FUNCTION "TE-SS" : VOID	// FC 11
AUTHOR : SIMATIC
FAMILY : EA_DIS
NAME : TE_SS
VERSION : 3.0
BEGIN
// (block stored without names or comments; labels and parameter names are numbered)
NETWORK
TITLE =
      L     0;
      L     #PARAM22;
      ==I;
      JC    M001;
      T     MW 214;
      L     MB 214;
      T     LW 10;
      OPN   DB [LW 10];
      L     MB 215;
      SLW   3;
      LAR1;
      L     DBW [AR1,P#0.0];
      T     MB 227;
M001: L     #PARAM20;
      T     MW 214;
      L     MB 214;
      T     LW 10;
      OPN   DB [LW 10];
      L     #PARAM20;
      T     MW 214;
      L     MB 215;
      SLW   3;
      LAR1;
      L     DBW [AR1,P#0.0];
      T     MW 200;
      L     DBW [AR1,P#2.0];
      T     MW 202;
      L     DBW [AR1,P#4.0];
      T     MW 204;
      L     DBW [AR1,P#10.0];
      T     MW 208;
      L     DBW [AR1,P#12.0];
      T     MW 210;
      L     DBW [AR1,P#14.0];
      T     MW 212;
      L     DBW [AR1,P#16.0];
      T     MW 206;
      A     #PARAM1;
      A     M 204.7;
      =     M 203.2;
      A     #PARAM1;
      AN    M 204.7;
      =     M 202.0;
      A     #PARAM2;
      =     M 202.1;
      A     #PARAM3;
      AN    M 203.3;
      =     M 211.5;
      A     #PARAM3;
      =     M 203.3;
      A     #PARAM4;
      AN    M 203.0;
      =     M 211.7;
      A     #PARAM4;
      =     M 203.0;
      A     #PARAM8;
      AN    M 203.1;
      =     M 211.6;
      A     #PARAM8;
      =     M 203.1;
      A     #PARAM9;
      AN    M 203.4;
      =     M 211.4;
      A     #PARAM9;
      =     M 203.4;
      A     #PARAM10;
      =     M 202.2;
      A     #PARAM11;
      =     M 203.5;
      A     #PARAM7;
      =     M 213.0;
      A     #PARAM6;
      =     M 210.1;
      A     #PARAM13;
      =     M 210.7;
      A     #PARAM14;
      =     M 210.6;
      A     #PARAM15;
      =     M 210.5;
      A     #PARAM16;
      =     M 210.4;
      A     #PARAM17;
      =     M 210.3;
      A     #PARAM18;
      =     M 210.2;
      A     #PARAM19;
      =     M 200.4;
      A     #PARAM12;
      =     M 210.0;
      A     #PARAM5;
      =     M 203.6;
NETWORK
TITLE =
      A     M 210.7;
      AN    M 210.6;
      =     M 212.7;
      AN    M 210.7;
      A     M 210.6;
      =     M 212.5;
      A     M 210.5;
      AN    M 210.4;
      =     M 212.6;
      AN    M 210.5;
      A     M 210.4;
      =     M 212.4;
NETWORK
TITLE =
      A     M 227.3;
      AN    M 202.5;
      =     M 211.3;
      A     M 227.3;
      =     M 202.5;
      A     M 227.2;
      AN    M 202.6;
      =     M 211.2;
      A     M 227.2;
      =     M 202.6;
NETWORK
TITLE =
      A     M 203.1;
      A     M 210.1;
      AN    M 203.0;
      AN    M 203.6;
      =     M 218.7;
      A     M 203.0;
      A     M 210.1;
      AN    M 203.6;
      =     M 219.7;
      A     M 227.2;
      A     M 227.1;
      AN    M 227.3;
      AN    M 227.0;
      AN    M 219.7;
      AN    M 203.6;
      =     M 218.5;
      A     M 227.3;
      A     M 227.1;
      AN    M 227.0;
      AN    M 218.7;
      AN    M 203.6;
      =     M 219.5;
      A     M 203.4;
      AN    M 203.3;
      AN    M 219.7;
      AN    M 203.6;
      AN    M 227.0;
      AN    M 219.5;
      =     M 218.3;
      A     M 203.3;
      AN    M 218.7;
      AN    M 218.5;
      AN    M 203.6;
      AN    M 227.0;
      =     M 219.3;
      A     M 218.7;
      O     M 218.5;
      O     M 218.3;
      =     M 212.3;
      A     M 219.7;
      O     M 219.5;
      O     M 219.3;
      =     M 212.1;
      A     M 211.6;
      A     M 218.7;
      O;
      A     M 211.2;
      A     M 218.5;
      O;
      A     M 211.4;
      A     M 218.3;
      =     M 212.2;
      A     M 211.7;
      A     M 219.7;
      O;
      A     M 211.3;
      A     M 219.5;
      O;
      A     M 211.5;
      A     M 219.3;
      =     M 212.0;
NETWORK
TITLE =
      A     M 211.6;
      O     M 211.2;
      =     M 213.4;
      A     M 211.7;
      O     M 211.3;
      =     M 213.5;
      A     M 203.6;
      O     M 227.0;
      =     M 213.7;
NETWORK
TITLE =
      A     M 212.7;
      O     M 213.7;
      O     M 212.3;
      R     M 211.1;
      R     M 211.0;
      A     M 203.2;
      S     M 211.1;
      A     M 202.0;
      S     M 211.0;
      A     M 212.6;
      O     M 213.7;
      O     M 212.1;
      R     M 213.1;
      A     M 203.5;
      S     M 213.1;
NETWORK
TITLE =
      A     M 203.1;
      A     M 210.1;
      O(;
      A     M 227.2;
      A     M 227.1;
      );
      O     M 203.4;
      =     M 213.2;
      A     M 203.0;
      A     M 210.1;
      O(;
      A     M 227.3;
      A     M 227.1;
      );
      O     M 203.3;
      =     M 213.3;
      A     M 213.2;
      O     M 203.5;
      ON    M 202.1;
      A     M 213.3;
      A     M 212.5;
      O(;
      A     M 213.3;
      O     M 203.2;
      O     M 202.0;
      ON    M 202.2;
      A     M 213.2;
      A     M 212.4;
      );
      O(;
      A     M 203.2;
      O     M 202.0;
      A     M 203.5;
      A     M 212.5;
      );
      =     M 201.1;
NETWORK
TITLE =
      L     0;
      L     MW 206;
      >=I;
      JC    M002;
      AN    "M 1.3";
      JC    M002;
      L     MW 206;
      L     1;
      -I;
      T     MW 206;
      L     MB 207;
      T     DBW [AR1,P#16.0];
M002: NOP   0;
NETWORK
TITLE =
      L     MB 205;
      T     MB 209;
      L     0;
      >I;
      JC    M006;
      A     M 212.7;
      A     M 212.4;
      AN    M 204.5;
      O;
      A     M 212.7;
      A     M 212.4;
      A     M 204.5;
      AN    M 210.3;
      L     1;
      JC    M005;
      A     M 212.6;
      A     M 212.5;
      AN    M 204.6;
      O;
      A     M 212.6;
      A     M 212.5;
      A     M 204.6;
      AN    M 210.2;
      L     9;
      JC    M005;
      A     M 212.0;
      A     M 202.1;
      AN    M 213.1;
      O     M 211.1;
      O     M 211.0;
      L     10;
      JC    M003;
      AN    M 212.2;
      ON    M 202.2;
      AN    M 213.1;
      JC    M004;
      L     2;
M003: T     MB 209;
      L     DBW [AR1,P#6.0];
      T     MW 206;
      L     MW 206;
      T     DBW [AR1,P#16.0];
      JU    M006;
M004: L     0;
M005: T     MB 209;
M006: NOP   0;
NETWORK
TITLE =
      L     MB 205;
      L     1;
      <>I;
      JC    M008;
      A     M 212.6;
      O     M 212.5;
      L     14;
      JC    M007;
      A     M 211.0;
      O     M 211.1;
      JC    M008;
      AN    M 212.2;
      ON    M 202.2;
      AN    M 213.1;
      JC    M008;
      L     DBW [AR1,P#6.0];
      T     MW 206;
      L     MW 206;
      T     DBW [AR1,P#16.0];
      L     2;
M007: T     MB 209;
M008: NOP   0;
NETWORK
TITLE =
      L     MB 205;
      L     2;
      <>I;
      JC    M014;
      A     M 212.0;
      A     M 202.1;
      AN    M 213.1;
      O     M 211.0;
      O     M 211.1;
      L     12;
      JC    M009;
      A     M 212.5;
      L     4;
      JC    M012;
      A     M 213.7;
      AN    M 213.1;
      O     M 200.4;
      O;
      AN    M 212.3;
      AN    M 213.0;
      AN    M 213.1;
      L     0;
      JC    M013;
      AN    M 210.2;
      L     6;
      JC    M013;
      L     MW 206;
      L     0;
      <>I;
      JC    M014;
      L     3;
      T     MB 209;
      JU    M014;
M009: T     MB 209;
      L     DBW [AR1,P#6.0];
      JU    M011;
M010: L     DBW [AR1,P#8.0];
M011: T     MW 206;
      T     DBW [AR1,P#16.0];
      JU    M014;
M012: T     MB 209;
      JU    M010;
M013: T     MB 209;
      L     0;
      JU    M011;
M014: NOP   0;
NETWORK
TITLE =
      L     MB 205;
      L     3;
      <>I;
      JC    M017;
      A     M 211.1;
      O     M 200.4;
      O;
      A     M 213.7;
      AN    M 213.1;
      O;
      AN    M 213.0;
      AN    M 212.3;
      AN    M 213.1;
      O;
      A     M 212.0;
      A     M 202.1;
      AN    M 213.1;
      L     0;
      JC    M016;
      A     M 212.7;
      A     M 213.5;
      L     1;
      JC    M016;
      A     M 212.5;
      A     M 213.4;
      L     4;
      JC    M015;
      A     M 210.2;
      L     6;
      JC    M017;
M015: T     MB 209;
      L     DBW [AR1,P#8.0];
      T     MW 206;
      L     MW 206;
      T     DBW [AR1,P#16.0];
      JU    M017;
M016: T     MB 209;
M017: NOP   0;
NETWORK
TITLE =
      L     MB 205;
      L     4;
      <>I;
      JC    M021;
      A     M 212.0;
      A     M 202.1;
      AN    M 213.1;
      O     M 211.0;
      O     M 211.1;
      L     10;
      JC    M018;
      A     M 212.6;
      AN    M 204.6;
      O;
      A     M 212.6;
      A     M 204.6;
      AN    M 210.2;
      L     9;
      JC    M020;
      A     M 213.7;
      AN    M 213.1;
      O     M 200.4;
      O;
      AN    M 212.3;
      AN    M 213.0;
      AN    M 213.1;
      L     0;
      JC    M020;
      AN    M 210.2;
      L     6;
      JC    M020;
      L     MW 206;
      L     0;
      <>I;
      JC    M021;
      L     5;
      T     MB 209;
      JU    M021;
M018: T     MB 209;
      L     DBW [AR1,P#6.0];
M019: T     MW 206;
      L     MW 206;
      T     DBW [AR1,P#16.0];
      JU    M021;
M020: T     MB 209;
      L     0;
      JU    M019;
M021: NOP   0;
NETWORK
TITLE =
      L     MB 205;
      L     5;
      <>I;
      JC    M024;
      A     M 213.7;
      O     M 200.4;
      O;
      AN    M 213.0;
      AN    M 212.3;
      AN    M 213.1;
      L     0;
      JC    M023;
      A     M 212.6;
      AN    M 204.6;
      A     M 213.4;
      O;
      A     M 212.6;
      A     M 204.6;
      AN    M 210.2;
      A     M 213.4;
      L     9;
      JC    M023;
      A     M 211.1;
      O;
      A     M 212.0;
      A     M 202.1;
      AN    M 213.1;
      L     10;
      JC    M022;
      A     M 210.2;
      L     6;
      JC    M024;
M022: T     MB 209;
      L     DBW [AR1,P#6.0];
      T     MW 206;
      L     MW 206;
      T     DBW [AR1,P#16.0];
      JU    M024;
M023: T     MB 209;
M024: NOP   0;
NETWORK
TITLE =
      L     MB 205;
      L     6;
      <>I;
      JC    M025;
      AN    M 213.5;
      AN    M 213.4;
      L     0;
      JC    M025;
      T     MB 209;
M025: NOP   0;
NETWORK
TITLE =
      L     MB 205;
      L     9;
      <>I;
      JC    M027;
      A     M 212.7;
      O     M 212.4;
      O     M 200.4;
      L     6;
      JC    M026;
      AN    M 211.0;
      AN    M 211.1;
      A(;
      AN    M 212.0;
      ON    M 202.1;
      O     M 213.1;
      );
      JC    M027;
      L     DBW [AR1,P#6.0];
      T     MW 206;
      L     MW 206;
      T     DBW [AR1,P#0.0];
      L     10;
M026: T     MB 209;
M027: NOP   0;
NETWORK
TITLE =
      L     MB 205;
      L     10;
      <>I;
      JC    M033;
      A     M 212.2;
      A     M 202.2;
      O     M 213.1;
      AN    M 211.0;
      AN    M 211.1;
      L     4;
      JC    M028;
      A     M 212.4;
      L     12;
      JC    M031;
      A     M 213.7;
      AN    M 211.1;
      AN    M 211.0;
      O     M 200.4;
      O;
      AN    M 212.1;
      AN    M 213.0;
      AN    M 211.1;
      AN    M 211.0;
      L     0;
      JC    M032;
      AN    M 210.3;
      L     14;
      JC    M032;
      L     MW 206;
      L     0;
      <>I;
      JC    M033;
      L     11;
      T     MB 209;
      JU    M033;
M028: T     MB 209;
      L     DBW [AR1,P#6.0];
      JU    M030;
M029: L     DBW [AR1,P#8.0];
M030: T     MW 206;
      L     MW 206;
      T     DBW [AR1,P#16.0];
      JU    M033;
M031: T     MB 209;
      JU    M029;
M032: T     MB 209;
      L     0;
      JU    M030;
M033: NOP   0;
NETWORK
TITLE =
      L     MB 205;
      L     11;
      <>I;
      JC    M036;
      A     M 200.4;
      O;
      A     M 213.7;
      AN    M 211.1;
      AN    M 211.0;
      O;
      AN    M 213.0;
      AN    M 212.1;
      AN    M 211.1;
      AN    M 211.0;
      O;
      A     M 212.2;
      A     M 202.2;
      AN    M 211.1;
      AN    M 211.0;
      L     0;
      JC    M035;
      A     M 212.6;
      A     M 213.4;
      L     9;
      JC    M035;
      A     M 212.4;
      A     M 213.5;
      L     12;
      JC    M034;
      A     M 210.3;
      L     14;
      JC    M036;
M034: T     MB 209;
      L     DBW [AR1,P#8.0];
      T     MW 206;
      L     MW 206;
      T     DBW [AR1,P#16.0];
      JU    M036;
M035: T     MB 209;
M036: NOP   0;
NETWORK
TITLE =
      L     MB 205;
      L     12;
      <>I;
      JC    M040;
      A     M 212.2;
      A     M 202.2;
      O     M 213.1;
      AN    M 211.0;
      AN    M 211.1;
      L     2;
      JC    M037;
      A     M 212.7;
      AN    M 204.5;
      O;
      A     M 212.7;
      A     M 204.5;
      AN    M 210.3;
      =     M 228.0;
      A     M 228.0;
      A     M 211.1;
      L     6;
      JC    M039;
      A     M 228.0;
      L     1;
      JC    M039;
      A     M 213.7;
      AN    M 211.1;
      AN    M 211.0;
      O     M 200.4;
      O;
      AN    M 212.1;
      AN    M 213.0;
      AN    M 211.1;
      AN    M 211.0;
      L     0;
      JC    M039;
      AN    M 210.3;
      L     14;
      JC    M039;
      L     MW 206;
      L     0;
      <>I;
      JC    M040;
      L     13;
      T     MB 209;
      JU    M040;
M037: T     MB 209;
      L     DBW [AR1,P#6.0];
M038: T     MW 206;
      L     MW 206;
      T     DBW [AR1,P#16.0];
      JU    M040;
M039: T     MB 209;
      L     0;
      JU    M038;
M040: NOP   0;
NETWORK
TITLE =
      L     MB 205;
      L     13;
      <>I;
      JC    M043;
      A     M 213.7;
      O     M 200.4;
      O;
      AN    M 213.0;
      AN    M 212.1;
      AN    M 211.1;
      AN    M 211.0;
      L     0;
      JC    M042;
      A     M 212.7;
      AN    M 204.5;
      A     M 213.5;
      O;
      A     M 212.7;
      A     M 204.5;
      AN    M 210.3;
      A     M 213.5;
      L     1;
      JC    M042;
      A     M 212.2;
      A     M 202.2;
      AN    M 211.1;
      AN    M 211.0;
      L     2;
      JC    M041;
      A     M 210.3;
      L     14;
      JC    M043;
M041: T     MB 209;
      L     DBW [AR1,P#6.0];
      T     MW 206;
      L     MW 206;
      T     DBW [AR1,P#16.0];
      JU    M043;
M042: T     MB 209;
M043: NOP   0;
NETWORK
TITLE =
      L     MB 205;
      L     14;
      <>I;
      JC    M044;
      AN    M 213.5;
      AN    M 213.4;
      L     0;
      JC    M044;
      T     MB 209;
M044: NOP   0;
NETWORK
TITLE =
      L     MB 209;
      T     MB 205;
      L     15;
      <I;
      A(;
      +     -7;
      <>I;
      );
      A(;
      +     -1;
      <>I;
      );
      AN    "M 0.7";
      JC    M045;
      L     0;
      T     MB 205;
M045: NOP   0;
NETWORK
TITLE =
      A     M 212.6;
      A     M 212.7;
      O;
      AN    M 212.6;
      AN    M 212.4;
      O;
      AN    M 212.7;
      AN    M 212.5;
      =     M 200.7;
      AN    M 210.2;
      AN    M 210.3;
      =     M 202.7;
      A     M 212.6;
      AN    M 210.2;
      =     M 200.5;
      A     M 212.7;
      AN    M 210.3;
      =     M 200.6;
      AN    M 209.0;
      A     M 209.1;
      A     M 209.2;
      AN    M 200.7;
      =     M 228.0;
      AN    M 209.3;
      A     M 228.0;
      =     M 200.2;
      A     M 209.3;
      A     M 228.0;
      =     M 200.3;
      A     M 209.0;
      A(;
      A     M 209.1;
      AN    M 209.2;
      O;
      AN    M 209.1;
      A     M 209.2;
      );
      AN    M 200.7;
      AN    M 202.7;
      =     M 228.0;
      A     M 228.0;
      AN    M 209.3;
      =     M 200.1;
      A     M 228.0;
      A     M 209.3;
      =     M 200.0;
NETWORK
TITLE =
      A     M 201.1;
      =     M 203.7;
      A     M 209.0;
      A     M 209.1;
      A     M 209.2;
      O     M 200.4;
      O     M 200.3;
      O     M 200.2;
      O     M 200.1;
      O     M 200.0;
      O     M 200.7;
      O     M 202.7;
      =     M 201.0;
      A(;
      A     M 209.1;
      AN    M 209.2;
      O;
      AN    M 209.1;
      A     M 209.2;
      );
      AN    M 209.0;
      =     M 228.0;
      A     M 228.0;
      A     M 209.3;
      =     M 201.4;
      A     M 200.0;
      O     M 200.3;
      AN    M 200.7;
      AN    M 202.7;
      =     M 201.2;
      A     M 212.7;
      AN    M 204.5;
      O;
      A     M 212.7;
      A     M 204.5;
      AN    M 210.3;
      =     M 201.3;
      =     M 202.4;
      =     #PARAM24;
      A     M 228.0;
      AN    M 209.3;
      =     M 201.7;
      A     M 200.1;
      O     M 200.2;
      AN    M 200.7;
      AN    M 202.7;
      =     M 201.5;
      A     M 212.6;
      AN    M 204.6;
      O;
      A     M 212.6;
      AN    M 210.2;
      A     M 204.6;
      =     M 201.6;
      =     M 202.3;
      =     #PARAM25;
NETWORK
TITLE =
      A     M 201.0;
      O     M 203.7;
      AN    M 201.1;
      =     #PARAM26;
      A     M 201.0;
      A     "M 1.6";
      O     M 203.7;
      O     #PARAM12;
      =     #PARAM29;
      A     M 201.7;
      A     "M 1.5";
      O;
      A     M 201.5;
      A     "M 1.6";
      O     M 201.6;
      O     #PARAM12;
      =     #PARAM28;
      A     M 201.4;
      A     "M 1.5";
      O;
      A     M 201.2;
      A     "M 1.6";
      O     M 201.3;
      O     #PARAM12;
      =     #PARAM27;
NETWORK
TITLE =
      A(;
      A     M 209.1;
      AN    M 209.2;
      O;
      AN    M 209.1;
      A     M 209.2;
      );
      AN    M 209.3;
      =     #PARAM31;
      A(;
      A     M 209.1;
      AN    M 209.2;
      O;
      AN    M 209.1;
      A     M 209.2;
      );
      A     M 209.3;
      =     #PARAM30;
      L     MW 200;
      T     DBW [AR1,P#0.0];
      L     MW 202;
      T     DBW [AR1,P#2.0];
      L     MW 204;
      T     DBW [AR1,P#4.0];
      L     MW 208;
      T     DBW [AR1,P#10.0];
      L     MW 210;
      T     DBW [AR1,P#12.0];
      L     MW 212;
      T     DBW [AR1,P#14.0];
      L     MW 206;
      T     DBW [AR1,P#16.0];
      L     0;
      L     #PARAM23;
      ==I;
      JC    M048;
      T     MW 216;
      T     MW 240;
      L     MB 216;
      SLW   3;
      LAR1;
      L     DBW [AR1,P#0.0];
      T     MW 242;
      L     MW 240;
      SLW   12;
      SRW   12;
      T     MW 240;
      L     8;
      L     MB 241;
      >I;
      JC    M046;
      +     -8;
      SLW   8;
      INC   242;
      JU    M047;
M046: SLW   8;
      INC   243;
M047: T     MW 244;
      L     MB 244;
      L     MB 245;
      SLW   3;
      OW;
      LAR2;
      A     M 201.0;
      O     M 203.3;
      =     M [AR2,P#0.0];
      L     MB 217;
      SLW   3;
      LAR1;
      L     MW 242;
      T     DBW [AR1,P#0.0];
M048: L     0;
      L     #PARAM21;
      ==I;
      BEC;
      T     MW 216;
      L     MB 216;
      T     LW 10;
      OPN   DB [LW 10];
      L     MB 217;
      SLW   3;
      LAR1;
      L     MW 200;
      T     DBW [AR1,P#0.0];
      L     MW 202;
      T     DBW [AR1,P#2.0];
END_FUNCTION

FUNCTION "TE-REK" : VOID	// FC 12
AUTHOR : SIMATIC
FAMILY : SIMATIC
NAME : TE_REK
VERSION : 3.0
BEGIN
// (block stored without names or comments; labels and parameter names are numbered)
NETWORK
TITLE =
      L     0;
      L     #PARAM20;
      ==I;
      JC    M001;
      T     MW 212;
      L     MB 212;
      T     LW 10;
      OPN   DB [LW 10];
      L     MB 213;
      SLW   3;
      LAR1;
      L     DBW [AR1,P#2.0];
M001: T     MW 210;
      L     #PARAM18;
      T     MW 214;
      L     MB 214;
      T     LW 10;
      OPN   DB [LW 10];
      L     MB 215;
      SLW   3;
      LAR1;
      L     DBW [AR1,P#0.0];
      T     MW 200;
      L     DBW [AR1,P#2.0];
      T     MW 202;
      A     #PARAM1;
      =     M 203.1;
      A     #PARAM2;
      =     M 200.4;
      A     #PARAM3;
      AN    M 202.7;
      =     M 210.0;
      A     #PARAM3;
      =     M 202.7;
      A     #PARAM4;
      AN    M 200.2;
      =     M 210.1;
      A     #PARAM4;
      =     M 200.2;
      A     #PARAM6;
      AN    M 200.3;
      =     M 210.3;
      A     #PARAM6;
      =     M 200.3;
      A     #PARAM7;
      AN    M 202.6;
      =     M 210.2;
      A     #PARAM7;
      =     M 202.6;
      A     #PARAM8;
      =     M 200.5;
      A     #PARAM9;
      =     M 203.0;
      A     #PARAM10;
      =     M 210.7;
      A     #PARAM5;
      =     M 202.5;
      A     #PARAM11;
      AN    M 200.0;
      =     M 210.4;
      A     #PARAM11;
      =     M 200.0;
      A     #PARAM12;
      AN    M 200.1;
      =     M 210.5;
      A     #PARAM12;
      =     M 200.1;
      A     #PARAM13;
      AN    M 202.4;
      =     M 210.6;
      A     #PARAM13;
      =     M 202.4;
      AN    #PARAM14;
      =     M 200.6;
      A     #PARAM15;
      =     M 203.3;
NETWORK
TITLE =
      A     M 211.0;
      AN    M 202.3;
      =     M 211.5;
      A     M 211.0;
      =     M 202.3;
      A     M 211.2;
      AN    M 202.1;
      =     M 211.6;
      A     M 211.2;
      =     M 202.1;
      A     M 211.3;
      AN    M 202.2;
      =     M 211.7;
      A     M 211.3;
      =     M 202.2;
NETWORK
TITLE =
      AN    M 200.7;
      AN    M 201.5;
      S     M 200.7;
      A     "´1´";
      R     M 201.7;
      R     M 201.6;
NETWORK
TITLE =
      A     M 202.7;
      A     M 202.5;
      O;
      A     M 202.1;
      A     M 211.1;
      O;
      A     M 200.2;
      =     M 202.0;
      A     M 202.6;
      A     M 202.5;
      O;
      A     M 202.2;
      A     M 211.1;
      O;
      A     M 200.3;
      =     M 203.6;
NETWORK
TITLE =
      AN    M 200.7;
      JC    M005;
      AN    M 203.1;
      JC    M002;
      L     MW 214;
      +     5;
      T     MW 216;
      +     -2;
      T     MW 218;
      L     DBW [AR1,P#10.0];
      T     DBW [AR1,P#6.0];
      JU    M005;
M002: AN    M 203.0;
      JC    M003;
      L     MW 214;
      +     6;
      T     MW 216;
      +     -3;
      T     MW 218;
      L     DBW [AR1,P#12.0];
      T     DBW [AR1,P#6.0];
      JU    M008;
M003: A     M 211.5;
      A     M 211.1;
      AN    M 202.4;
      O;
      A     M 210.6;
      A     M 202.5;
      AN    M 211.0;
      S     M 201.7;
      A     M 210.5;
      AN    M 200.0;
      O     M 201.7;
      O     M 211.5;
      R     M 200.7;
      S     M 201.5;
      R     M 210.5;
      R     M 211.5;
      R     M 210.6;
      A     M 202.0;
      AN    M 203.6;
      A     M 200.4;
      S     M 203.5;
      AN    M 202.0;
      R     M 203.5;
      A     M 203.6;
      AN    M 202.0;
      A     M 200.5;
      S     M 203.4;
      AN    M 203.6;
      R     M 203.4;
      AN    M 203.5;
      JC    M006;
      L     MW 214;
      +     2;
      T     MW 216;
      L     DBW [AR1,P#4.0];
      T     MW 206;
      SLW   6;
      SRW   6;
      L     DBB [AR1,P#4.0];
      SRW   2;
      +I;
      L     1000;
      TAK;
      >I;
      JC    M004;
      TAK;
M004: T     MW 204;
      L     MB 206;
      SRW   2;
      SLW   10;
      OW;
      T     DBW [AR1,P#4.0];
      L     MW 214;
      +     3;
      T     MW 216;
      L     DBW [AR1,P#6.0];
      L     MW 204;
      -I;
      T     DBW [AR1,P#6.0];
M005: JU    M008;
M006: AN    M 203.4;
      JC    M009;
      L     MW 214;
      +     2;
      T     MW 216;
      L     DBW [AR1,P#4.0];
      T     MW 206;
      SLW   6;
      SRW   6;
      L     DBB [AR1,P#4.0];
      SRW   2;
      +I;
      L     1000;
      TAK;
      >I;
      JC    M007;
      TAK;
M007: T     MW 204;
      L     MB 206;
      SRW   2;
      SLW   10;
      OW;
      T     DBW [AR1,P#4.0];
      L     MW 214;
      +     3;
      T     MW 216;
      L     DBW [AR1,P#6.0];
      L     MW 204;
      +I;
      T     DBW [AR1,P#6.0];
M008: JU    M010;
M009: L     MW 214;
      +     2;
      T     MW 216;
      L     DBB [AR1,P#4.0];
      SRW   2;
      SLW   10;
      T     DBW [AR1,P#4.0];
      L     0;
      L     #PARAM20;
      ==I;
      JC    M010;
      T     MW 212;
      L     MW 214;
      +     8;
      T     MW 216;
      L     DBW [AR1,P#16.0];
      T     LD 0;
      L     MB 212;
      T     LW 10;
      OPN   DB [LW 10];
      L     MB 213;
      SLW   3;
      LAR1;
      L     LD 0;
      L     DBW [AR1,P#0.0];
      ==I;
      T     LD 0;
      L     MB 214;
      T     LW 10;
      OPN   DB [LW 10];
      JC    M010;
      L     MB 215;
      SLW   3;
      LAR1;
      L     LD 0;
      T     DBW [AR1,P#16.0];
      L     MW 214;
      +     3;
      T     MW 216;
      L     LD 0;
      T     DBW [AR1,P#6.0];
M010: NOP   0;
NETWORK
TITLE =
      AN    M 201.5;
      JC    M013;
      AN    M 203.1;
      JC    M011;
      L     MW 214;
      +     5;
      T     MW 216;
      +     -2;
      T     MW 218;
      L     MB 215;
      SLW   3;
      LAR1;
      L     DBW [AR1,P#10.0];
      T     DBW [AR1,P#6.0];
      JU    M012;
M011: AN    M 203.0;
      JC    M012;
      L     MW 214;
      +     6;
      T     MW 216;
      +     -3;
      T     MW 218;
      L     MB 215;
      SLW   3;
      LAR1;
      L     DBW [AR1,P#12.0];
      T     DBW [AR1,P#6.0];
M012: A     M 211.5;
      A     M 211.1;
      AN    M 202.4;
      O;
      A     M 210.6;
      A     M 202.5;
      AN    M 211.0;
      S     M 201.6;
      A     M 210.4;
      AN    M 200.1;
      AN    M 202.4;
      AN    M 202.3;
      O     M 211.5;
      O     M 201.6;
      O     M 200.6;
      O     "M 0.6";
      O     M 203.3;
      S     M 200.7;
      R     M 201.5;
      A     M 200.7;
      O     M 203.0;
      O     M 203.1;
      JC    M013;
      L     #PARAM16;
      T     MW 216;
      L     MB 216;
      T     LW 10;
      OPN   DB [LW 10];
      L     MB 217;
      SLW   3;
      LAR1;
      L     DBD [AR1,P#0.0];
      T     LD 0;
      L     MB 214;
      T     LW 10;
      OPN   DB [LW 10];
      L     MW 214;
      +     3;
      T     MW 216;
      L     MB 215;
      SLW   3;
      LAR1;
      L     LW 8;
      L     LD 0;
      T     DBD [AR1,P#18.0];
M013: NOP   0;
NETWORK
TITLE =
      L     MW 214;
      +     3;
      T     MW 216;
      +     4;
      T     MW 218;
      L     MB 215;
      SLW   3;
      LAR1;
      L     DBW [AR1,P#6.0];
      L     DBW [AR1,P#14.0];
      ==I;
      T     MW 222;
      JC    M019;
      <=I;
      JC    M016;
      AN    M 200.5;
      AN    M 203.0;
      JC    M019;
      TAK;
      T     MW 224;
      L     MW 214;
      +     6;
      T     MW 216;
      L     DBW [AR1,P#12.0];
      L     DBW [AR1,P#10.0];
      -I;
      SRW   3;
      L     MW 222;
      +I;
      L     MW 224;
      <=I;
      TAK;
      JC    M014;
      TAK;
M014: T     MW 222;
      L     MW 214;
      +     6;
      T     MW 216;
      L     DBW [AR1,P#12.0];
      L     MW 222;
      >I;
      JC    M015;
      L     MW 214;
      +     3;
      T     MW 216;
      L     DBW [AR1,P#12.0];
      T     DBW [AR1,P#6.0];
M015: NOP   0;
      T     DBW [AR1,P#14.0];
      T     MW 222;
      L     MW 218;
      +     2;
      T     MW 218;
      TAK;
      L     MW 222;
      L     1;
      *I;
      DTR;
      T     DBD [AR1,P#18.0];
      JU    M019;
M016: ==I;
      JC    M019;
      AN    M 200.4;
      AN    M 203.1;
      JC    M019;
      TAK;
      T     MW 224;
      L     MW 214;
      +     6;
      T     MW 216;
      L     DBW [AR1,P#12.0];
      L     DBW [AR1,P#10.0];
      -I;
      SRW   3;
      L     MW 222;
      TAK;
      -I;
      L     MW 224;
      >=I;
      TAK;
      JC    M017;
      TAK;
M017: T     MW 222;
      L     MW 214;
      +     5;
      T     MW 216;
      L     DBW [AR1,P#10.0];
      L     MW 222;
      <I;
      JC    M018;
      L     MW 214;
      +     3;
      T     MW 216;
      L     DBW [AR1,P#10.0];
      T     DBW [AR1,P#6.0];
M018: NOP   0;
      T     DBW [AR1,P#14.0];
      T     MW 222;
      L     1;
      *I;
      DTR;
      T     DBD [AR1,P#18.0];
M019: NOP   0;
NETWORK
TITLE =
      A(;
      A     M 203.0;
      O     M 203.1;
      ON    M 200.5;
      ON    M 200.4;
      A     M 201.5;
      );
      O(;
      A(;
      O     M 202.4;
      O     M 202.3;
      );
      A(;
      O     M 200.6;
      O     M 203.3;
      );
      );
      O(;
      A     M 203.0;
      ON    M 200.4;
      A     M 202.0;
      A     M 200.7;
      );
      O(;
      A     M 203.1;
      ON    M 200.5;
      A     M 203.6;
      A     M 200.7;
      );
      =     M 201.3;
      A     M 203.5;
      O     M 203.4;
      O     M 203.0;
      O     M 203.1;
      =     M 203.7;
      =     M 203.2;
NETWORK
TITLE =
// (network holds code this reader does not know; not shown)
END_FUNCTION

FUNCTION "TE-TS" : VOID	// FC 13
AUTHOR : SIMATIC
FAMILY : EA_DIS
NAME : TE_TS
VERSION : 3.0
BEGIN
// (block stored without names or comments; labels and parameter names are numbered)
NETWORK
TITLE =
      L     0;
      L     #PARAM9;
      ==I;
      JC    M001;
      T     MW 212;
      L     MB 212;
      T     LW 10;
      OPN   DB [LW 10];
      L     MB 213;
      SLW   3;
      LAR1;
      L     DBW [AR1,P#0.0];
      T     MB 207;
M001: OPN   #PARAM6;
      L     #PARAM7;
      T     MW 212;
      L     MB 213;
      SLW   3;
      LAR1;
      L     DBW [AR1,P#0.0];
      T     MW 200;
      A     #PARAM1;
      AN    M 201.5;
      =     M 203.5;
      A     #PARAM1;
      =     M 201.5;
      A     #PARAM2;
      AN    M 201.6;
      =     M 203.6;
      A     #PARAM2;
      =     M 201.6;
      A     #PARAM3;
      AN    M 201.4;
      =     M 203.4;
      A     #PARAM3;
      =     M 201.4;
      A     #PARAM4;
      =     M 201.3;
      A     #PARAM5;
      =     M 200.7;
NETWORK
TITLE =
      A     M 207.0;
      A     M 207.1;
      AN    M 200.0;
      =     M 203.0;
      A     M 207.0;
      =     M 200.0;
NETWORK
TITLE =
      A     M 207.3;
      AN    M 200.3;
      =     M 203.3;
      A     M 207.3;
      =     M 200.3;
NETWORK
TITLE =
      A     M 207.2;
      AN    M 200.2;
      =     M 203.2;
      A     M 207.2;
      =     M 200.2;
NETWORK
TITLE =
      A     M 203.0;
      A     M 207.1;
      A     M 201.7;
      =     M 203.1;
      A     M 203.0;
      A     M 207.1;
      AN    M 201.7;
      =     M 203.7;
      A     M 203.6;
      A     M 201.3;
      A     M 201.7;
      =     M 202.0;
      A     M 203.6;
      A     M 201.3;
      AN    M 201.7;
      =     M 202.1;
NETWORK
TITLE =
      A     M 200.2;
      A     M 207.1;
      O;
      A     M 201.7;
      A     M 200.0;
      A     M 207.1;
      O;
      A     M 201.7;
      A     M 201.6;
      A     M 201.3;
      O     M 201.5;
      =     M 200.5;
      A     M 200.3;
      A     M 207.1;
      O;
      AN    M 201.7;
      A     M 200.0;
      A     M 207.1;
      O;
      AN    M 201.7;
      A     M 201.6;
      A     M 201.3;
      O     M 201.4;
      =     M 200.6;
NETWORK
TITLE =
      A(;
      A     M 203.3;
      AN    M 200.2;
      O     M 203.7;
      O     M 202.1;
      O     M 201.4;
      );
      S     M 201.7;
      A(;
      A     M 203.2;
      AN    M 200.3;
      O     M 203.1;
      O     M 202.0;
      );
      AN    M 201.4;
      O     M 201.5;
      R     M 201.7;
NETWORK
TITLE =
      A     M 201.7;
      =     M 201.2;
      =     #PARAM11;
      AN    M 201.7;
      =     M 201.1;
      =     #PARAM12;
      A     M 200.6;
      A     M 200.5;
      =     M 201.0;
NETWORK
TITLE =
      A     M 201.0;
      O     M 200.7;
      =     #PARAM14;
      A     M 201.1;
      O     M 200.7;
      =     #PARAM13;
      A     M 201.2;
      O     M 200.7;
      =     #PARAM15;
NETWORK
TITLE =
      L     MW 200;
      T     DBW [AR1,P#0.0];
      L     0;
      L     #PARAM10;
      ==I;
      JC    M004;
      T     MW 212;
      T     MW 220;
      L     MB 212;
      SLW   3;
      LAR1;
      L     DBW [AR1,P#2.0];
      T     MW 208;
      L     MW 220;
      SLW   12;
      SRW   12;
      T     MW 220;
      L     8;
      L     MB 221;
      >I;
      JC    M002;
      +     -8;
      SLW   8;
      INC   208;
      JU    M003;
M002: SLW   8;
      INC   209;
M003: T     MW 210;
      L     MB 210;
      L     MB 211;
      SLW   3;
      OW;
      LAR2;
      A     M 201.0;
      =     M [AR2,P#0.0];
      L     MB 212;
      SLW   3;
      LAR1;
      L     MW 208;
      T     DBW [AR1,P#2.0];
M004: L     0;
      L     #PARAM8;
      ==I;
      JC    M005;
      T     MW 214;
      L     MB 214;
      T     LW 10;
      OPN   DB [LW 10];
      L     MB 215;
      SLW   3;
      LAR1;
      L     MW 200;
      T     DBW [AR1,P#0.0];
M005: NOP   0;
END_FUNCTION

FUNCTION "TE-VW3/3" : VOID	// FC 14
AUTHOR : SIMATIC
FAMILY : EA_DIS
NAME : TE_VW3_3
VERSION : 3.0
BEGIN
// (block stored without names or comments; labels and parameter names are numbered)
NETWORK
TITLE =
      L     0;
      L     #PARAM14;
      ==I;
      JC    M001;
      T     MW 212;
      L     MB 212;
      T     LW 10;
      OPN   DB [LW 10];
      L     MB 213;
      SLW   3;
      LAR1;
      L     DBW [AR1,P#0.0];
      T     MB 203;
M001: L     #PARAM12;
      T     MW 214;
      L     MB 214;
      T     LW 10;
      OPN   DB [LW 10];
      L     MB 215;
      SLW   3;
      LAR1;
      L     DBW [AR1,P#0.0];
      T     MW 200;
      L     DBW [AR1,P#2.0];
      T     MB 202;
      A     #PARAM1;
      =     M 200.0;
      A     #PARAM2;
      AN    M 201.7;
      =     M 204.5;
      A     #PARAM2;
      =     M 201.7;
      A     #PARAM3;
      AN    M 200.1;
      =     M 205.4;
      A     #PARAM3;
      =     M 200.1;
      A     #PARAM4;
      =     M 200.3;
      A     #PARAM5;
      AN    M 200.2;
      =     M 204.6;
      A     #PARAM5;
      =     M 200.2;
      A     #PARAM6;
      AN    M 200.4;
      =     M 205.5;
      A     #PARAM6;
      =     M 200.4;
      A     #PARAM7;
      =     M 200.6;
      A     #PARAM8;
      AN    M 200.5;
      =     M 204.7;
      A     #PARAM8;
      =     M 200.5;
      A     #PARAM9;
      AN    M 200.7;
      =     M 205.6;
      A     #PARAM9;
      =     M 200.7;
      A     #PARAM10;
      =     M 201.6;
      A     #PARAM11;
      =     M 201.5;
NETWORK
TITLE =
      A     M 203.0;
      AN    M 202.0;
      =     M 204.0;
      A     M 203.0;
      =     M 202.0;
      A     M 203.1;
      AN    M 202.1;
      =     M 204.1;
      A     M 203.1;
      =     M 202.1;
      A     M 203.2;
      AN    M 202.2;
      =     M 204.2;
      A     M 203.2;
      =     M 202.2;
NETWORK
TITLE =
      A(;
      A     M 205.4;
      A     M 201.6;
      O;
      A     M 204.0;
      AN    M 200.4;
      AN    M 200.7;
      O;
      A     M 204.5;
      AN    M 200.4;
      AN    M 200.7;
      AN    M 203.1;
      AN    M 203.2;
      );
      A     M 200.0;
      =     M 202.5;
      A(;
      A     M 205.5;
      A     M 201.6;
      O;
      A     M 204.1;
      AN    M 200.1;
      AN    M 200.7;
      O;
      A     M 204.6;
      AN    M 200.1;
      AN    M 200.7;
      AN    M 203.0;
      AN    M 203.2;
      );
      A     M 200.3;
      =     M 202.6;
      A(;
      A     M 205.6;
      A     M 201.6;
      O;
      A     M 204.2;
      AN    M 200.4;
      AN    M 200.1;
      O;
      A     M 204.7;
      AN    M 200.4;
      AN    M 200.1;
      AN    M 203.1;
      AN    M 203.0;
      );
      A     M 200.6;
      =     M 202.7;
NETWORK
TITLE =
      AN    M 201.1;
      AN    M 201.2;
      S     M 201.0;
      A     "´1´";
      S     M 201.3;
      R     M 201.4;
NETWORK
TITLE =
      AN    M 201.0;
      JC    M002;
      A     M 202.6;
      S     M 201.1;
      R     M 201.0;
      A     M 202.7;
      S     M 201.2;
      R     M 201.0;
M002: NOP   0;
NETWORK
TITLE =
      AN    M 201.1;
      JC    M003;
      A     M 202.5;
      S     M 201.0;
      R     M 201.1;
      A     M 202.7;
      S     M 201.2;
      R     M 201.1;
M003: NOP   0;
NETWORK
TITLE =
      AN    M 201.2;
      JC    M004;
      A     M 202.6;
      S     M 201.1;
      R     M 201.2;
      A     M 202.5;
      S     M 201.0;
      R     M 201.2;
M004: NOP   0;
NETWORK
TITLE =
      A     M 201.0;
      =     #PARAM15;
      A     M 201.1;
      =     #PARAM16;
      A     M 201.2;
      =     #PARAM17;
      A     M 201.0;
      O     M 201.5;
      =     #PARAM18;
      A     M 201.1;
      O     M 201.5;
      =     #PARAM19;
      A     M 201.2;
      O     M 201.5;
      =     #PARAM20;
      L     MW 200;
      T     DBW [AR1,P#0.0];
      L     MW 202;
      T     DBW [AR1,P#2.0];
      L     0;
      L     #PARAM13;
      ==I;
      BEC;
      T     MW 216;
      L     MB 216;
      T     LW 10;
      OPN   DB [LW 10];
      L     MB 217;
      SLW   3;
      LAR1;
      L     MB 201;
      T     DBW [AR1,P#0.0];
END_FUNCTION

FUNCTION "TE-KO" : VOID	// FC 15
AUTHOR : SIMATIC
FAMILY : EA_DIS
NAME : TE_KO
VERSION : 0.0
BEGIN
// (block stored without names or comments; labels and parameter names are numbered)
NETWORK
TITLE =
      L     0;
      L     #PARAM18;
      ==I;
      JC    M001;
      T     MW 214;
      L     MB 214;
      T     LW 10;
      OPN   DB [LW 10];
      L     MB 215;
      SLW   3;
      LAR1;
      L     DBW [AR1,P#0.0];
      T     MB 230;
M001: L     #PARAM16;
      T     MW 214;
      L     MB 214;
      T     LW 10;
      OPN   DB [LW 10];
      L     #PARAM16;
      T     MW 214;
      L     MB 215;
      SLW   3;
      LAR1;
      L     DBW [AR1,P#8.0];
      T     MB 203;
      L     DBW [AR1,P#12.0];
      T     MB 209;
      L     DBW [AR1,P#16.0];
      T     MB 212;
      A     #PARAM1;
      =     M 202.0;
      =     #PARAM22;
      A     #PARAM2;
      =     M 203.4;
      A     #PARAM3;
      AN    M 212.2;
      =     M 220.3;
      A     #PARAM3;
      =     M 212.2;
      A     #PARAM4;
      AN    M 203.2;
      =     M 220.1;
      A     #PARAM4;
      =     M 203.2;
      A     #PARAM5;
      =     M 202.2;
      =     #PARAM23;
      A     #PARAM6;
      AN    M 203.0;
      =     M 221.6;
      A     #PARAM6;
      =     M 203.0;
      A     #PARAM7;
      AN    M 212.0;
      =     M 220.2;
      A     #PARAM7;
      =     M 212.0;
      A     #PARAM9;
      AN    M 203.1;
      =     M 221.7;
      A     #PARAM9;
      =     M 203.1;
      A     #PARAM10;
      =     M 202.3;
      =     #PARAM28;
      A     #PARAM11;
      AN    M 203.3;
      =     M 220.0;
      A     #PARAM11;
      =     M 203.3;
      A     #PARAM12;
      AN    M 212.3;
      =     M 220.4;
      A     #PARAM12;
      =     M 212.3;
      A     #PARAM13;
      =     M 203.5;
      A     #PARAM14;
      =     M 202.1;
      =     #PARAM29;
      A     #PARAM8;
      =     M 221.5;
      A     #PARAM15;
      =     M 221.4;
NETWORK
TITLE =
      A     M 230.0;
      AN    M 212.4;
      =     M 220.5;
      A     M 230.0;
      =     M 212.4;
      A     M 230.4;
      AN    M 212.6;
      =     M 220.6;
      A     M 230.4;
      =     M 212.6;
      A     M 230.5;
      AN    M 212.7;
      =     M 220.7;
      A     M 230.5;
      =     M 212.7;
NETWORK
TITLE =
      A(;
      A     M 220.2;
      A     M 221.5;
      O;
      A     M 220.5;
      A     M 230.1;
      );
      =     M 232.1;
      AN    M 232.1;
      AN    M 221.7;
      AN    M 221.6;
      JC    M002;
      A     M 221.7;
      AN    M 203.0;
      O     M 232.1;
      AN    M 209.0;
      S     M 209.0;
      R     M 232.1;
      A     M 221.6;
      O     M 232.1;
      A     M 209.0;
      R     M 209.0;
M002: NOP   0;
NETWORK
TITLE =
      A(;
      A     M 220.4;
      A     M 221.5;
      O;
      A     M 220.7;
      A     M 230.1;
      AN    M 230.4;
      O;
      A     M 220.0;
      AN    M 203.2;
      AN    M 230.4;
      );
      AN    M 212.2;
      =     M 221.3;
NETWORK
TITLE =
      A(;
      A     M 220.3;
      A     M 221.5;
      O;
      A     M 220.6;
      A     M 230.1;
      AN    M 212.3;
      O;
      A     M 220.1;
      AN    M 212.3;
      AN    M 230.5;
      );
      =     M 221.2;
NETWORK
TITLE =
      A     M 212.3;
      A     M 221.5;
      O;
      A     M 230.5;
      A     M 230.1;
      O;
      A     M 203.3;
      =     M 221.1;
      A     M 212.2;
      A     M 221.5;
      O;
      A     M 230.4;
      A     M 230.1;
      O;
      A     M 203.2;
      =     M 221.0;
      A(;
      A(;
      AN    M 203.5;
      O     M 202.0;
      A     M 221.0;
      A     M 203.4;
      );
      A     M 221.1;
      );
      O(;
      A(;
      AN    M 203.4;
      O     M 202.1;
      A     M 221.1;
      A     M 203.5;
      );
      A     M 221.0;
      );
      O(;
      A     M 203.0;
      A     M 203.1;
      );
      =     M 200.1;
NETWORK
TITLE =
      A     M 209.0;
      =     #PARAM26;
      JC    M003;
      R     M 212.1;
      R     M 212.5;
      R     M 209.3;
      R     M 209.4;
M003: NOP   0;
NETWORK
TITLE =
      AN    M 209.0;
      =     #PARAM25;
      JC    M004;
      A     M 221.2;
      A     M 203.4;
      AN    M 202.1;
      O     M 202.0;
      S     M 212.5;
      R     M 212.1;
      A     M 221.3;
      A     M 203.5;
      O     M 202.1;
      AN    M 202.0;
      S     M 212.1;
      R     M 212.5;
M004: NOP   0;
NETWORK
TITLE =
      AN    M 212.1;
      A     M 209.2;
      R     M 209.4;
      R     M 200.7;
      JC    M005;
      S     M 200.7;
      AN    M 212.1;
      S     M 209.2;
      A     M 212.1;
      R     M 209.2;
M005: A     M 209.4;
      =     M 202.5;
NETWORK
TITLE =
      AN    M 212.5;
      A     M 209.1;
      R     M 209.3;
      R     M 200.6;
      JC    M006;
      S     M 200.6;
      AN    M 212.5;
      S     M 209.1;
      A     M 212.5;
      R     M 209.1;
M006: A     M 209.3;
      =     M 202.4;
NETWORK
TITLE =
      A(;
      A     M 212.3;
      A     M 221.5;
      O;
      A     M 230.5;
      A     M 230.1;
      );
      A     M 203.5;
      A     M 209.0;
      =     M 200.5;
      =     #PARAM30;
      A(;
      A     M 212.2;
      A     M 221.5;
      O;
      A     M 230.4;
      A     M 230.1;
      );
      A     M 203.4;
      A     M 209.0;
      =     M 200.4;
      =     #PARAM21;
NETWORK
TITLE =
      A     M 230.0;
      A     M 230.1;
      O;
      A     M 221.5;
      A     #PARAM7;
      =     M 232.0;
      A     M 209.0;
      A     M 232.0;
      =     M 200.3;
      AN    M 209.0;
      A     M 232.0;
      =     M 200.2;
NETWORK
TITLE =
      A     M 200.7;
      A     M 202.2;
      =     M 203.7;
      A     M 200.6;
      A     M 202.3;
      =     M 203.6;
NETWORK
TITLE =
      A     M 202.5;
      O     M 202.4;
      O     M 203.7;
      O     M 203.6;
      =     M 200.0;
      A     M 202.5;
      O     M 203.7;
      =     M 201.5;
      A     M 202.4;
      O     M 203.6;
      =     M 201.2;
      A     M 200.7;
      AN    M 202.3;
      =     M 201.7;
      A     M 200.6;
      AN    M 202.2;
      =     M 201.4;
      A     M 200.7;
      A     M 202.3;
      =     M 201.6;
      A     M 200.6;
      A     M 202.2;
      =     M 201.3;
      A     M 209.0;
      =     M 201.1;
      AN    M 209.0;
      =     M 201.0;
NETWORK
TITLE =
      A     M 200.6;
      =     #PARAM24;
      A     M 200.7;
      =     #PARAM27;
      O(;
      A     "M 0.5";
      A     M 201.4;
      O;
      A     "M 1.6";
      A     M 201.2;
      O;
      O     M 201.3;
      O     M 221.4;
      );
      =     #PARAM31;
      A     M 201.0;
      O     M 221.4;
      =     #PARAM32;
      A     M 200.0;
      A     "M 1.6";
      O     M 200.1;
      O     M 221.4;
      =     #PARAM33;
      A     M 201.1;
      O     M 221.4;
      =     #PARAM34;
      O(;
      A     M 201.7;
      A     "M 0.5";
      O;
      A     M 201.5;
      A     "M 1.6";
      O;
      O     M 201.6;
      O     M 221.4;
      );
      =     #PARAM35;
      L     MW 200;
      T     DBW [AR1,P#6.0];
      L     MW 202;
      T     DBW [AR1,P#8.0];
      L     MW 208;
      T     DBW [AR1,P#12.0];
      L     MW 210;
      T     DBW [AR1,P#14.0];
      L     MB 212;
      T     DBW [AR1,P#16.0];
      L     MW 220;
      T     DBW [AR1,P#18.0];
      L     0;
      L     #PARAM20;
      ==I;
      JC    M009;
      T     MW 216;
      T     MW 240;
      L     MB 216;
      SLW   3;
      LAR1;
      L     DBW [AR1,P#0.0];
      T     MW 242;
      L     MW 240;
      SLW   12;
      SRW   12;
      T     MW 240;
      L     8;
      L     MB 241;
      >I;
      JC    M007;
      +     -8;
      SLW   8;
      INC   242;
      JU    M008;
M007: SLW   8;
      INC   243;
M008: T     MW 244;
      L     MB 244;
      L     MB 245;
      SLW   3;
      OW;
      LAR2;
      A     M 201.0;
      O     M 203.3;
      =     M [AR2,P#0.0];
      L     MB 217;
      SLW   3;
      LAR1;
      L     MW 242;
      T     DBW [AR1,P#0.0];
M009: L     0;
      L     #PARAM17;
      ==I;
      BEC;
      T     MW 222;
      L     MB 222;
      T     LW 10;
      OPN   DB [LW 10];
      L     MB 223;
      SLW   3;
      LAR1;
      L     MW 200;
      T     DBW [AR1,P#6.0];
      L     MW 202;
      T     DBW [AR1,P#8.0];
END_FUNCTION

FUNCTION "TE-VW2/2" : VOID	// FC 16
AUTHOR : SIMATIC
FAMILY : EA_DIS
NAME : TE_VW2_2
VERSION : 3.0
BEGIN
// (block stored without names or comments; labels and parameter names are numbered)
NETWORK
TITLE =
      L     0;
      L     #PARAM11;
      ==I;
      JC    M001;
      T     MW 212;
      L     MB 212;
      T     LW 10;
      OPN   DB [LW 10];
      L     MB 213;
      SLW   3;
      LAR1;
      L     DBW [AR1,P#0.0];
      T     MB 203;
M001: L     #PARAM9;
      T     MW 214;
      L     MB 214;
      T     LW 10;
      OPN   DB [LW 10];
      L     MB 215;
      SLW   3;
      LAR1;
      L     DBW [AR1,P#0.0];
      T     MW 200;
      L     DBW [AR1,P#2.0];
      T     MB 202;
      A     #PARAM1;
      =     M 200.0;
      A     #PARAM2;
      AN    M 201.7;
      =     M 204.5;
      A     #PARAM2;
      =     M 201.7;
      A     #PARAM3;
      AN    M 200.1;
      =     M 205.4;
      A     #PARAM3;
      =     M 200.1;
      A     #PARAM4;
      =     M 200.3;
      A     #PARAM5;
      AN    M 200.2;
      =     M 204.6;
      A     #PARAM5;
      =     M 200.2;
      A     #PARAM6;
      AN    M 200.4;
      =     M 205.5;
      A     #PARAM6;
      =     M 200.4;
      A     #PARAM7;
      =     M 201.6;
      A     #PARAM8;
      =     M 201.5;
NETWORK
TITLE =
      A     M 203.0;
      AN    M 202.0;
      =     M 204.0;
      A     M 203.0;
      =     M 202.0;
      A     M 203.1;
      AN    M 202.1;
      =     M 204.1;
      A     M 203.1;
      =     M 202.1;
NETWORK
TITLE =
      A(;
      A     M 205.4;
      A     M 201.6;
      O;
      A     M 204.0;
      AN    M 200.4;
      O;
      A     M 204.5;
      AN    M 200.4;
      AN    M 203.1;
      );
      A     M 200.0;
      =     M 202.5;
      A(;
      A     M 205.5;
      A     M 201.6;
      O;
      A     M 204.1;
      AN    M 200.1;
      O;
      A     M 204.6;
      AN    M 200.1;
      AN    M 203.0;
      );
      A     M 200.3;
      =     M 202.6;
NETWORK
TITLE =
      AN    M 201.1;
      S     M 201.0;
      A     "´1´";
      R     M 201.3;
      S     M 201.4;
NETWORK
TITLE =
      AN    M 201.0;
      JC    M002;
      A     M 202.6;
      S     M 201.1;
      R     M 201.0;
M002: NOP   0;
NETWORK
TITLE =
      AN    M 201.1;
      JC    M003;
      A     M 202.5;
      S     M 201.0;
      R     M 201.1;
M003: NOP   0;
NETWORK
TITLE =
      A     M 201.0;
      =     #PARAM12;
      A     M 201.1;
      =     #PARAM13;
      A     M 201.0;
      O     M 201.5;
      =     #PARAM14;
      A     M 201.1;
      O     M 201.5;
      =     #PARAM15;
      L     MW 200;
      T     DBW [AR1,P#0.0];
      L     MB 202;
      T     DBW [AR1,P#2.0];
      L     0;
      L     #PARAM10;
      ==I;
      BEC;
      T     MW 216;
      L     MB 216;
      T     LW 10;
      OPN   DB [LW 10];
      L     MB 217;
      SLW   3;
      LAR1;
      L     MB 201;
      T     DBW [AR1,P#0.0];
NETWORK
TITLE =
END_FUNCTION

FUNCTION "TE-VW2/1" : VOID	// FC 17
AUTHOR : SIMATIC
FAMILY : EA_DIS
NAME : TE_VW2_1
VERSION : 3.0
BEGIN
// (block stored without names or comments; labels and parameter names are numbered)
NETWORK
TITLE =
      L     0;
      L     #PARAM10;
      ==I;
      JC    M001;
      T     MW 212;
      L     MB 212;
      T     LW 10;
      OPN   DB [LW 10];
      L     MB 213;
      SLW   3;
      LAR1;
      L     DBW [AR1,P#0.0];
      T     MB 203;
M001: L     #PARAM8;
      T     MW 214;
      L     MB 214;
      T     LW 10;
      OPN   DB [LW 10];
      L     MB 215;
      SLW   3;
      LAR1;
      L     DBW [AR1,P#0.0];
      T     MW 200;
      L     DBW [AR1,P#2.0];
      T     MB 202;
      A     #PARAM1;
      =     M 200.0;
      A     #PARAM2;
      AN    M 201.7;
      =     M 204.5;
      A     #PARAM2;
      =     M 201.7;
      A     #PARAM3;
      AN    M 200.1;
      =     M 204.3;
      A     #PARAM3;
      =     M 200.1;
      A     #PARAM4;
      =     M 200.3;
      A     #PARAM5;
      AN    M 200.2;
      =     M 204.6;
      A     #PARAM5;
      =     M 200.2;
      A     #PARAM6;
      =     M 201.6;
      A     #PARAM7;
      =     M 201.5;
NETWORK
TITLE =
      A     M 203.0;
      AN    M 202.0;
      =     M 204.0;
      A     M 203.0;
      =     M 202.0;
NETWORK
TITLE =
      A     M 204.3;
      A     M 201.6;
      O;
      A     M 204.0;
      AN    M 200.1;
      =     M 202.5;
NETWORK
TITLE =
      AN    M 201.1;
      S     M 201.0;
      A     "´1´";
      R     M 201.3;
      R     M 201.4;
NETWORK
TITLE =
      AN    M 201.0;
      JC    M002;
      A     M 202.5;
      O     M 204.6;
      A     M 200.3;
      S     M 201.1;
      R     M 201.0;
      R     M 202.5;
M002: NOP   0;
NETWORK
TITLE =
      AN    M 201.1;
      JC    M003;
      A     M 202.5;
      O     M 204.5;
      A     M 200.0;
      S     M 201.0;
      R     M 201.1;
      R     M 202.5;
M003: NOP   0;
NETWORK
TITLE =
      A     M 201.0;
      =     #PARAM11;
      A     M 201.1;
      =     #PARAM12;
      A     M 201.0;
      O     M 201.5;
      =     #PARAM13;
      A     M 201.1;
      O     M 201.5;
      =     #PARAM14;
      L     MW 200;
      T     DBW [AR1,P#0.0];
      L     MB 202;
      T     DBW [AR1,P#2.0];
      L     0;
      L     #PARAM9;
      ==I;
      BEC;
      T     MW 216;
      L     MB 216;
      T     LW 10;
      OPN   DB [LW 10];
      L     MB 217;
      SLW   3;
      LAR1;
      L     MB 201;
      T     DBW [AR1,P#0.0];
NETWORK
TITLE =
END_FUNCTION

FUNCTION "TE_READ_RTM" : VOID	// FC 18
AUTHOR : SIMATIC
FAMILY : S7_300
NAME : TE_RTM
VERSION : 0.1
BEGIN
// (block stored without names or comments; labels and parameter names are numbered)
NETWORK
TITLE =
      OPN   #PARAM2;
      L     #PARAM3;
      T     MW 224;
      L     MB 225;
      SLW   3;
      LAR1;
      L     DBW [AR1,P#0.0];
      T     MW 210;
      L     DBW [AR1,P#2.0];
      T     MW 212;
      L     DBW [AR1,P#4.0];
      T     MW 214;
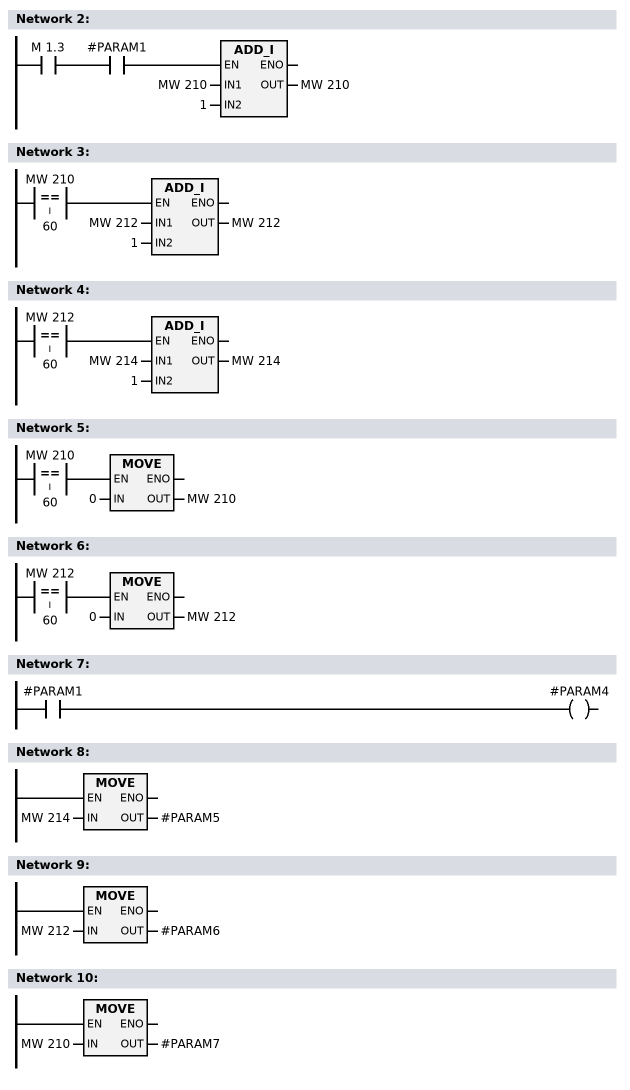
NETWORK
TITLE =
      A     "M 1.3";
      A     #PARAM1;
      JNB   M001;
      L     MW 210;
      L     1;
      +I;
      T     MW 210;
M001: NOP   0;
NETWORK
TITLE =
      A(;
      L     MW 210;
      L     60;
      ==I;
      );
      JNB   M002;
      L     MW 212;
      L     1;
      +I;
      T     MW 212;
M002: NOP   0;
NETWORK
TITLE =
      A(;
      L     MW 212;
      L     60;
      ==I;
      );
      JNB   M003;
      L     MW 214;
      L     1;
      +I;
      T     MW 214;
M003: NOP   0;
NETWORK
TITLE =
      A(;
      L     MW 210;
      L     60;
      ==I;
      );
      JNB   M004;
      L     0;
      T     MW 210;
M004: NOP   0;
NETWORK
TITLE =
      A(;
      L     MW 212;
      L     60;
      ==I;
      );
      JNB   M005;
      L     0;
      T     MW 212;
M005: NOP   0;
NETWORK
TITLE =
      A     #PARAM1;
      =     #PARAM4;
NETWORK
TITLE =
      L     MW 214;
      T     #PARAM5;
      NOP   0;
NETWORK
TITLE =
      L     MW 212;
      T     #PARAM6;
      NOP   0;
NETWORK
TITLE =
      L     MW 210;
      T     #PARAM7;
      NOP   0;
NETWORK
TITLE =
      L     MB 225;
      SLW   3;
      LAR1;
      T     DBW [AR1,P#0.0];
      L     MW 210;
      T     DBW [AR1,P#0.0];
      L     MW 212;
      T     DBW [AR1,P#2.0];
      L     MW 214;
      T     DBW [AR1,P#4.0];
END_FUNCTION

FUNCTION "TE-TAK" : VOID	// FC 29
AUTHOR : SIMATIC
FAMILY : EA_DIS
NAME : TE_TAKT
VERSION : 3.0
BEGIN
// (block stored without names or comments; labels and parameter names are numbered)
NETWORK
TITLE =
      OPN   #PARAM2;
      L     #PARAM1;
      L     0;
      <>I;
      JC    M005;
      L     DBB 33;
      T     MB 203;
      L     DBW 28;
      T     MW 200;
      A     M 201.0;
      S     M 203.0;
      L     MB 201;
      L     0;
      <>I;
      JC    M001;
      S     M 203.1;
      S     M 203.2;
      JU    M002;
M001: +     5;
      ==I;
      S     M 203.1;
      JU    M004;
M002: A     M 200.0;
      S     M 203.3;
      L     MB 200;
      L     0;
      <>I;
      JC    M003;
      S     M 203.6;
      S     M 203.5;
      JU    M004;
M003: +     30;
      <>I;
      JC    M004;
      S     M 203.5;
M004: L     MB 203;
      T     DBB 33;
      L     DBB 29;
      +     1;
      T     DBB 29;
      L     10;
      <I;
      BEC;
      L     0;
      T     DBB 29;
      L     DBB 28;
      +     1;
      T     DBB 28;
      L     60;
      <I;
      BEC;
      L     0;
      T     DBB 28;
      BEU;
M005: NOP   0;
NETWORK
TITLE =
// (network holds code this reader does not know; not shown)
NETWORK
TITLE =
      +     1;
      <>I;
      JC    M009;
      L     0;
      T     DBB 31;
M009: NOP   0;
NETWORK
TITLE =
END_FUNCTION

FUNCTION "TE-GRENZ" : VOID	// FC 36
AUTHOR : SIMATIC
FAMILY : EA_DIS
NAME : TE_GRENZ
VERSION : 3.0
BEGIN
// (block stored without names or comments; labels and parameter names are numbered)
NETWORK
TITLE =
      AN    #PARAM4;
      R     #PARAM5;
      R     #PARAM6;
      BEC;
      L     #PARAM1;
      L     DW#16#0;
      ==R;
      JC    M001;
      L     #PARAM1;
      L     #PARAM2;
      >=R;
      S     #PARAM5;
      R     #PARAM6;
      BEC;
      L     #PARAM1;
      L     #PARAM3;
      <R;
M001: R     #PARAM5;
      S     #PARAM6;
NETWORK
TITLE =
END_FUNCTION

FUNCTION "TE-RETTEN" : VOID	// FC 38
AUTHOR : SIMATIC
FAMILY : EA_DIS
NAME : TE_RET
VERSION : 3.0
BEGIN
// (block stored without names or comments; labels and parameter names are numbered)
NETWORK
TITLE =
      OPN   #PARAM1;
      LAR1  P#DBX 0.0;
      LAR2  P#M 200.0;
      L     28;
M001: T     DBW 60;
      L     MW [AR2,P#0.0];
      T     DBW [AR1,P#0.0];
      +AR1  P#2.0;
      +AR2  P#2.0;
      L     DBW 60;
      LOOP  M001;
END_FUNCTION

FUNCTION "TE-LADEN" : VOID	// FC 39
AUTHOR : SIMATIC
FAMILY : EA_DIS
NAME : TE_LADEN
VERSION : 3.0
BEGIN
// (block stored without names or comments; labels and parameter names are numbered)
NETWORK
TITLE =
      OPN   #PARAM1;
      LAR1  P#DBX 0.0;
      LAR2  P#M 200.0;
      L     28;
M001: T     DBW 60;
      L     DBW [AR1,P#0.0];
      T     MW [AR2,P#0.0];
      +AR1  P#2.0;
      +AR2  P#2.0;
      L     DBW 60;
      LOOP  M001;
END_FUNCTION

FUNCTION "TE-SCHALTER" : VOID	// FC 49
AUTHOR : SIMATIC
FAMILY : S7_300
NAME : ASL_MOD
VERSION : 0.0
BEGIN
// (block stored without names or comments; labels and parameter names are numbered)
NETWORK
TITLE =
      L     #PARAM2;
      T     MW 202;
      L     #PARAM3;
      T     MW 204;
      L     #PARAM4;
      T     MW 206;
      L     MB 202;
      T     LW 10;
      OPN   DB [LW 10];
      L     MB 203;
      SLW   3;
      LAR1;
      L     DBD [AR1,P#0.0];
      T     MD 210;
      AN    #PARAM1;
      JC    M001;
      L     MB 204;
      T     LW 10;
      OPN   DB [LW 10];
      L     MB 205;
      SLW   3;
      LAR1;
      L     DBD [AR1,P#0.0];
      T     MD 210;
M001: NOP   0;
      L     MB 206;
      T     LW 10;
      OPN   DB [LW 10];
      L     MB 207;
      SLW   3;
      LAR1;
      L     MD 210;
      T     DBD [AR1,P#0.0];
END_FUNCTION

FUNCTION "G7_STD_3" : VOID	// FC 72
AUTHOR : SIMATIC
FAMILY : S7GRAPH
NAME : SFMULTI
VERSION : 2.0
BEGIN
// (block stored without names or comments; labels and parameter names are numbered)
NETWORK
TITLE =
// (network holds code this reader does not know; not shown)
NETWORK
TITLE =
      L     DID [AR1,P#80.0];
      LAR2;
      L     DID [AR2,P#14.0];
      T     LD 30;
      L     DID [AR2,P#18.0];
      T     LD 40;
      L     DID [AR1,P#48.0];
      AD    DW#16#7FFFF;
      LAR2;
      AN    L 30.7;
      JC    M007;
      A     DIX [AR2,P#0.0];
      FP    DIX [AR1,P#7.4];
      S     DIX [AR1,P#11.4];
      +AR2  P#0.1;
M007: AN    L 30.6;
      JC    M008;
      A     DIX [AR2,P#0.0];
      FP    DIX [AR1,P#7.5];
      S     DIX [AR1,P#11.5];
      +AR2  P#0.1;
M008: AN    L 30.5;
      JC    M009;
      A     DIX [AR2,P#0.0];
      FP    DIX [AR1,P#9.3];
      S     DIX [AR1,P#13.3];
      +AR2  P#0.1;
M009: AN    L 30.4;
      JC    M010;
      A     DIX [AR2,P#0.0];
      FP    DIX [AR1,P#9.2];
      S     DIX [AR1,P#13.2];
      +AR2  P#0.1;
M010: AN    L 30.3;
      JC    M011;
      A     DIX [AR2,P#0.0];
      FP    DIX [AR1,P#6.4];
      S     DIX [AR1,P#10.4];
      +AR2  P#0.1;
M011: AN    L 30.2;
      JC    M012;
      A     DIX [AR2,P#0.0];
      FP    DIX [AR1,P#6.5];
      S     DIX [AR1,P#10.5];
      +AR2  P#0.1;
M012: AN    L 30.1;
      JC    M013;
      A     DIX [AR2,P#0.0];
      FP    DIX [AR1,P#7.6];
      X     DIX [AR1,P#11.6];
      =     DIX [AR1,P#11.6];
      +AR2  P#0.1;
M013: AN    L 30.0;
      JC    M014;
      A     DIX [AR2,P#0.0];
      FP    DIX [AR1,P#7.7];
      X     DIX [AR1,P#11.7];
      =     DIX [AR1,P#11.7];
      +AR2  P#0.1;
M014: AN    L 31.7;
      JC    M015;
      A     DIX [AR2,P#0.0];
      FP    DIX [AR1,P#8.0];
      X     DIX [AR1,P#12.0];
      =     DIX [AR1,P#12.0];
      +AR2  P#0.1;
M015: AN    L 31.6;
      JC    M016;
      A     DIX [AR2,P#0.0];
      FP    DIX [AR1,P#7.0];
      X     DIX [AR1,P#11.0];
      =     DIX [AR1,P#11.0];
      +AR2  P#0.1;
M016: AN    L 31.5;
      JC    M017;
      A     DIX [AR2,P#0.0];
      FP    DIX [AR1,P#7.1];
      X     DIX [AR1,P#11.1];
      =     DIX [AR1,P#11.1];
      +AR2  P#0.1;
M017: AN    L 31.4;
      JC    M018;
      A     DIX [AR2,P#0.0];
      FP    DIX [AR1,P#7.2];
      X     DIX [AR1,P#11.2];
      =     DIX [AR1,P#11.2];
      +AR2  P#0.1;
M018: AN    L 31.3;
      JC    M019;
      A     DIX [AR2,P#0.0];
      FP    DIX [AR1,P#7.3];
      X     DIX [AR1,P#11.3];
      =     DIX [AR1,P#11.3];
      +AR2  P#0.1;
M019: AN    L 31.2;
      JC    M020;
      A     DIX [AR2,P#0.0];
      FP    DIX [AR1,P#8.1];
      S     DIX [AR1,P#12.1];
      R     DIX [AR1,P#12.2];
      R     DIX [AR1,P#12.3];
      R     DIX [AR1,P#12.4];
      R     DIX [AR1,P#12.5];
      +AR2  P#0.1;
M020: AN    L 31.1;
      JC    M021;
      A     DIX [AR2,P#0.0];
      FP    DIX [AR1,P#8.2];
      R     DIX [AR1,P#12.1];
      S     DIX [AR1,P#12.2];
      R     DIX [AR1,P#12.3];
      R     DIX [AR1,P#12.4];
      R     DIX [AR1,P#12.5];
      +AR2  P#0.1;
M021: AN    L 31.0;
      JC    M022;
      A     DIX [AR2,P#0.0];
      FP    DIX [AR1,P#8.3];
      R     DIX [AR1,P#12.1];
      R     DIX [AR1,P#12.2];
      S     DIX [AR1,P#12.3];
      R     DIX [AR1,P#12.4];
      R     DIX [AR1,P#12.5];
      +AR2  P#0.1;
M022: AN    L 32.7;
      JC    M023;
      A     DIX [AR2,P#0.0];
      FP    DIX [AR1,P#8.4];
      S     DIX [AR1,P#12.4];
      +AR2  P#0.1;
M023: AN    L 32.6;
      JC    M024;
      A     DIX [AR2,P#0.0];
      FP    DIX [AR1,P#8.5];
      S     DIX [AR1,P#12.5];
      +AR2  P#0.1;
M024: AN    L 32.5;
      JC    M025;
      A     DIX [AR2,P#0.0];
      FP    DIX [AR1,P#6.0];
      =     L 29.1;
      S     DIX [AR1,P#10.0];
      R     DIX [AR1,P#10.2];
      R     DIX [AR1,P#10.3];
      R     DIX [AR1,P#10.1];
      +AR2  P#0.1;
      R     DIX [AR1,P#12.4];
      R     DIX [AR1,P#12.5];
      R     DIX [AR1,P#10.6];
      R     DIX [AR1,P#10.7];
      AN    L 31.2;
      AN    L 31.1;
      AN    L 31.0;
      A     L 29.1;
      S     DIX [AR1,P#12.1];
      R     DIX [AR1,P#12.2];
      R     DIX [AR1,P#12.3];
M025: AN    L 32.4;
      JC    M026;
      A     DIX [AR2,P#0.0];
      FP    DIX [AR1,P#6.2];
      =     L 29.1;
      R     DIX [AR1,P#10.0];
      S     DIX [AR1,P#10.2];
      R     DIX [AR1,P#10.3];
      R     DIX [AR1,P#10.1];
      +AR2  P#0.1;
      R     DIX [AR1,P#12.4];
      R     DIX [AR1,P#12.5];
      R     DIX [AR1,P#10.6];
      R     DIX [AR1,P#10.7];
      AN    L 31.2;
      AN    L 31.1;
      AN    L 31.0;
      A     L 29.1;
      S     DIX [AR1,P#12.1];
      R     DIX [AR1,P#12.2];
      R     DIX [AR1,P#12.3];
M026: AN    L 32.3;
      JC    M027;
      A     DIX [AR2,P#0.0];
      FP    DIX [AR1,P#6.3];
      =     L 29.1;
      R     DIX [AR1,P#10.0];
      R     DIX [AR1,P#10.2];
      S     DIX [AR1,P#10.3];
      R     DIX [AR1,P#10.1];
      +AR2  P#0.1;
      R     DIX [AR1,P#12.4];
      R     DIX [AR1,P#12.5];
      R     DIX [AR1,P#10.6];
      R     DIX [AR1,P#10.7];
      AN    L 31.2;
      AN    L 31.1;
      AN    L 31.0;
      A     L 29.1;
      S     DIX [AR1,P#12.1];
      R     DIX [AR1,P#12.2];
      R     DIX [AR1,P#12.3];
M027: AN    L 32.2;
      JC    M028;
      A     DIX [AR2,P#0.0];
      FP    DIX [AR1,P#6.1];
      =     L 29.1;
      R     DIX [AR1,P#10.0];
      R     DIX [AR1,P#10.2];
      R     DIX [AR1,P#10.3];
      S     DIX [AR1,P#10.1];
      +AR2  P#0.1;
      R     DIX [AR1,P#12.4];
      R     DIX [AR1,P#12.5];
      R     DIX [AR1,P#10.6];
      R     DIX [AR1,P#10.7];
      AN    L 31.2;
      AN    L 31.1;
      AN    L 31.0;
      A     L 29.1;
      R     DIX [AR1,P#12.1];
      R     DIX [AR1,P#12.2];
      S     DIX [AR1,P#12.3];
M028: AN    L 32.1;
      JC    M031;
      +AR2  P#1.7;
      TAR2;
      SRD   4;
      SLD   4;
      LAR2;
      AN    L 32.0;
      JC    M029;
      L     DIW [AR2,P#0.0];
      T     DIW [AR1,P#2.0];
      JU    M030;
M029: L     DIW [AR1,P#2.0];
      L     DIW [AR2,P#0.0];
      T     DIW [AR1,P#2.0];
      <>I;
      S     DIX [AR1,P#12.6];
M030: +AR2  P#2.0;
M031: AN    L 32.0;
      JC    M032;
      A     DIX [AR2,P#0.0];
      FP    DIX [AR1,P#8.6];
      S     DIX [AR1,P#12.6];
      +AR2  P#0.1;
M032: AN    L 33.7;
      JC    M033;
      A     DIX [AR2,P#0.0];
      FP    DIX [AR1,P#8.7];
      S     DIX [AR1,P#12.7];
      +AR2  P#0.1;
M033: AN    L 33.6;
      JC    M034;
      A     DIX [AR2,P#0.0];
      FP    DIX [AR1,P#9.0];
      S     DIX [AR1,P#13.0];
      +AR2  P#0.1;
M034: AN    L 33.5;
      JC    M035;
      A     DIX [AR2,P#0.0];
      FP    DIX [AR1,P#6.6];
      S     DIX [AR1,P#10.6];
      +AR2  P#0.1;
M035: AN    L 33.4;
      JC    M036;
      A     DIX [AR2,P#0.0];
      FP    DIX [AR1,P#6.7];
      S     DIX [AR1,P#10.7];
      +AR2  P#0.1;
M036: AN    L 33.3;
      JC    M037;
      A     DIX [AR2,P#0.0];
      FP    DIX [AR1,P#9.1];
      S     DIX [AR1,P#13.1];
M037: NOP   0;
NETWORK
TITLE =
      BLD   7;
      UC    "TIME_TCK";
      {     P#L 8.0 };
      BLD   8;
      L     LD 8;
      T     DID [AR1,P#22.0];
      A     DIX [AR1,P#11.7];
      JC    M038;
      L     DID [AR1,P#18.0];
      -D;
      T     DID [AR1,P#14.0];
      AD    DW#16#FFFFF000;
      JZ    M039;
M038: L     B#16#0;
      T     DID [AR1,P#14.0];
M039: L     DID [AR1,P#22.0];
      T     DID [AR1,P#18.0];
NETWORK
TITLE =
      L     DID [AR1,P#48.0];
      LAR2;
      L     DIW [AR1,P#52.0];
      T     LW 12;
      SET;
      S     DIX [AR1,P#27.5];
      AN    DIX [AR1,P#13.6];
      JC    M040;
      A     DIX [AR1,P#10.1];
      =     DIX [AR1,P#13.4];
M040: LAR1  LD 0;
      L     B#16#1;
      T     DIB [AR1,P#30.0];
      UC    FB [LW 12];
NETWORK
TITLE =
      LAR1  LD 4;
      L     DID [AR1,P#14.0];
      T     LW 22;
      CLR;
      LAR1  LD 0;
      L     DID [AR1,P#4.0];
      T     LD 8;
      LAR1;
      L     DIB [AR1,P#0.0];
      JU    M045;
M041: T     LB 16;
      +AR1  P#1.0;
      L     DIB [AR1,P#0.0];
      SLW   7;
      LAR2  LD 0;
      +AR2;
      +AR2;
      L     DID [AR2,P#4.0];
      L     LW 22;
      +D;
      <=D;
      JC    M042;
      L     DW#16#7FFFFFFF;
M042: T     DID [AR2,P#4.0];
      O     DIX [AR2,P#1.1];
      O     DIX [AR2,P#1.2];
      JC    M044;
      L     DID [AR2,P#8.0];
      L     LW 22;
      +D;
      <=D;
      JC    M043;
      L     DW#16#7FFFFFFF;
M043: T     DID [AR2,P#8.0];
M044: L     LB 16;
M045: LOOP  M041;
NETWORK
TITLE =
      LAR1  LD 4;
      L     DID [AR1,P#40.0];
      LAR1;
      SET;
      R     L 29.0;
      JU    M285;
M046: LAR1  LD 8;
      SET;
      S     L 29.0;
      JU    M285;
M047: LAR1  LD 4;
      L     DID [AR1,P#44.0];
      LAR2;
      L     B#16#1;
      T     DIB [AR2,P#0.0];
      L     DID [AR1,P#40.0];
      LAR2;
      L     B#16#1;
      T     DIB [AR2,P#0.0];
      L     DID [AR1,P#36.0];
      LAR2;
      L     B#16#1;
      T     DIB [AR2,P#0.0];
      LAR1  LD 8;
      L     B#16#0;
      JU    M251;
M048: NOP   0;
NETWORK
TITLE =
      LAR1  LD 4;
      AN    DIX [AR1,P#11.4];
      JC    M050;
      R     DIX [AR1,P#11.4];
      R     DIX [AR1,P#11.5];
      LAR1  LD 8;
      L     B#16#0;
      JU    M261;
M049: JU    M080;
M050: NOP   0;
NETWORK
TITLE =
      LAR1  LD 4;
      AN    DIX [AR1,P#11.5];
      JC    M056;
      R     DIX [AR1,P#11.5];
      R     DIX [AR1,P#26.4];
      R     DIX [AR1,P#26.5];
      R     DIX [AR1,P#26.6];
      R     DIX [AR1,P#26.7];
      R     DIX [AR1,P#27.0];
      R     DIX [AR1,P#26.3];
      LAR1  LD 8;
      L     B#16#1;
      JU    M261;
M051: LAR1  LD 0;
      L     DIW [AR1,P#28.0];
      SLD   3;
      LAR1;
      L     B#16#0;
      JU    M256;
M052: LAR1  LD 4;
      L     DID [AR1,P#40.0];
      LAR1;
      L     B#16#4;
      JU    M270;
M053: LAR1  LD 4;
      L     DID [AR1,P#36.0];
      T     LD 8;
      LAR1;
      L     B#16#3;
      JU    M270;
M054: LAR1  LD 8;
      L     B#16#1;
      JU    M251;
M055: JU    M080;
M056: NOP   0;
NETWORK
TITLE =
      LAR1  LD 4;
      AN    DIX [AR1,P#13.3];
      AN    DIX [AR1,P#13.2];
      JC    M060;
      A     DIX [AR1,P#13.3];
      R     DIX [AR1,P#26.1];
      R     DIX [AR1,P#26.2];
      R     DIX [AR1,P#26.0];
      R     DIX [AR1,P#26.4];
      R     DIX [AR1,P#26.5];
      R     DIX [AR1,P#26.6];
      R     DIX [AR1,P#26.7];
      R     DIX [AR1,P#27.0];
      R     DIX [AR1,P#26.3];
      LAR2  LD 0;
      L     DIW [AR2,P#18.0];
      SLD   3;
      T     LD 24;
      L     DIB [LD 24];
      JU    M059;
M057: T     LB 17;
      L     LD 24;
      +     L#8;
      T     LD 24;
      L     DIB [LD 24];
      SLW   7;
      LAR2  LD 0;
      +AR2;
      +AR2;
      A     DIX [AR1,P#13.2];
      S     DIX [AR2,P#0.3];
      AN    DIX [AR1,P#13.3];
      JC    M058;
      S     DIX [AR2,P#0.4];
      R     DIX [AR2,P#1.2];
      L     B#16#0;
      T     DID [AR2,P#8.0];
M058: L     LB 17;
M059: LOOP  M057;
      R     DIX [AR1,P#13.2];
M060: R     DIX [AR1,P#13.3];
NETWORK
TITLE =
      AN    DIX [AR1,P#10.4];
      AN    DIX [AR1,P#10.5];
      JC    M061;
      L     B#16#0;
      L     DIB [AR1,P#4.0];
      ==I;
      JC    M061;
      SLW   7;
      LAR2  LD 0;
      +AR2;
      +AR2;
      A     DIX [AR1,P#10.5];
      A(;
      O     DIX [AR2,P#1.1];
      O     DIX [AR2,P#1.2];
      );
      S     DIX [AR2,P#0.3];
      A     DIX [AR1,P#10.4];
      A(;
      O     DIX [AR2,P#1.1];
      O     DIX [AR2,P#1.2];
      );
      JCN   M061;
      S     DIX [AR2,P#0.4];
      R     DIX [AR2,P#1.2];
      L     B#16#0;
      T     DID [AR2,P#8.0];
M061: R     DIX [AR1,P#10.5];
      R     DIX [AR1,P#10.4];
NETWORK
TITLE =
      AN    DIX [AR1,P#12.4];
      JC    M064;
      L     B#16#0;
      L     DIB [AR1,P#4.0];
      ==I;
      JC    M064;
      L     B#16#2;
      L     DIB [AR1,P#4.0];
      >I;
      JC    M062;
      DEC   1;
      JU    M063;
M062: L     DID [AR1,P#80.0];
      LAR2;
      L     DIB [AR2,P#12.0];
M063: T     DIB [AR1,P#4.0];
      A     DIX [AR1,P#12.3];
      JC    M064;
      SLW   7;
      LAR2  LD 0;
      +AR2;
      +AR2;
      A     DIX [AR1,P#12.1];
      A     DIX [AR2,P#1.0];
      O;
      A     DIX [AR1,P#12.2];
      A(;
      O     DIX [AR2,P#1.1];
      O     DIX [AR2,P#1.2];
      );
M064: R     DIX [AR1,P#12.4];
NETWORK
TITLE =
      AN    DIX [AR1,P#12.5];
      JC    M066;
      L     B#16#0;
      L     DIB [AR1,P#4.0];
      ==I;
      JC    M066;
      L     DID [AR1,P#80.0];
      LAR2;
      L     DIB [AR2,P#12.0];
      L     DIB [AR1,P#4.0];
      INC   1;
      >=I;
      JC    M065;
      L     B#16#1;
M065: T     DIB [AR1,P#4.0];
      A     DIX [AR1,P#12.3];
      JC    M066;
      SLW   7;
      LAR2  LD 0;
      +AR2;
      +AR2;
      A     DIX [AR1,P#12.1];
      A     DIX [AR2,P#1.0];
      O;
      A     DIX [AR1,P#12.2];
      A(;
      O     DIX [AR2,P#1.1];
      O     DIX [AR2,P#1.2];
      );
M066: R     DIX [AR1,P#12.5];
NETWORK
TITLE =
      ON    DIX [AR1,P#10.1];
      ON    DIX [AR1,P#12.6];
      JC    M068;
      L     DIW [AR1,P#2.0];
      L     B#16#2;
      JU    M266;
M067: TAK;
      L     B#16#0;
      ==I;
      JC    M068;
      TAK;
      T     DIB [AR1,P#4.0];
M068: R     DIX [AR1,P#12.6];
NETWORK
TITLE =
      AN    DIX [AR1,P#10.1];
      R     DIX [AR1,P#12.7];
      AN    DIX [AR1,P#12.7];
      JC    M070;
      R     DIX [AR1,P#12.7];
      L     DIW [AR1,P#0.0];
      L     B#16#0;
      JU    M266;
M069: <>I;
      R     L 29.0;
      TAK;
      JC    M288;
M070: LAR1  LD 4;
      L     DID [AR1,P#68.0];
      T     LD 8;
      LAR1;
      LAR2  LD 0;
      L     DIB [AR2,P#26.0];
      SLW   3;
      +AR1;
      L     B#16#1;
      JU    M256;
M071: NOP   0;
NETWORK
TITLE =
      LAR1  LD 4;
      AN    DIX [AR1,P#10.1];
      R     DIX [AR1,P#13.0];
      AN    DIX [AR1,P#13.0];
      JC    M073;
      R     DIX [AR1,P#13.0];
      LAR2  LD 0;
      L     DID [AR2,P#4.0];
      LAR2;
      L     DIB [AR2,P#0.0];
      L     B#16#1;
      ==I;
      S     DIX [AR1,P#26.5];
      JC    M073;
      L     DIW [AR1,P#0.0];
      L     B#16#1;
      JU    M266;
M072: TAK;
      L     B#16#0;
      <>I;
      S     L 29.0;
      TAK;
      JC    M288;
M073: LAR1  LD 8;
      L     B#16#2;
      JU    M261;
M074: NOP   0;
NETWORK
TITLE =
      LAR1  LD 4;
      AN    DIX [AR1,P#10.6];
      JC    M077;
      L     B#16#0;
      L     DIB [AR1,P#5.0];
      ==I;
      JC    M077;
      L     B#16#2;
      L     DIB [AR1,P#5.0];
      >I;
      JC    M075;
      DEC   1;
      JU    M076;
M075: L     DID [AR1,P#80.0];
      LAR2;
      L     DIB [AR2,P#9.0];
M076: T     DIB [AR1,P#5.0];
      LAR2  LD 0;
      L     DIW [AR2,P#12.0];
      SLD   3;
      LAR2;
      TAK;
      SLW   7;
      +AR2;
      O(;
      O     DIX [AR1,P#10.0];
      O     DIX [AR1,P#10.3];
      A     DIX [AR2,P#0.0];
      );
      O(;
      O     DIX [AR1,P#10.1];
      O     DIX [AR1,P#10.2];
      A     DIX [AR2,P#0.1];
      );
M077: R     DIX [AR1,P#10.6];
NETWORK
TITLE =
      AN    DIX [AR1,P#10.7];
      JC    M079;
      L     B#16#0;
      L     DIB [AR1,P#5.0];
      ==I;
      JC    M079;
      L     DID [AR1,P#80.0];
      LAR2;
      L     DIB [AR2,P#9.0];
      L     DIB [AR1,P#5.0];
      INC   1;
      >=I;
      JC    M078;
      L     B#16#1;
M078: T     DIB [AR1,P#5.0];
      LAR2  LD 0;
      L     DIW [AR2,P#12.0];
      SLD   3;
      LAR2;
      TAK;
      SLW   7;
      +AR2;
      O(;
      O     DIX [AR1,P#10.0];
      O     DIX [AR1,P#10.3];
      A     DIX [AR2,P#0.0];
      );
      O(;
      O     DIX [AR1,P#10.1];
      O     DIX [AR1,P#10.2];
      A     DIX [AR2,P#0.1];
      );
M079: R     DIX [AR1,P#10.7];
NETWORK
TITLE =
M080: LAR1  LD 4;
      L     DID [AR1,P#68.0];
      LAR1;
      L     B#16#1;
      T     DIB [AR1,P#0.0];
      LAR2  LD 0;
      L     DIB [AR2,P#26.0];
      SLW   3;
      +AR1;
      TAK;
      T     DIB [AR1,P#0.0];
NETWORK
TITLE =
M081: SET;
      LAR1  LD 0;
      L     DIW [AR1,P#12.0];
      SLD   3;
      T     LD 8;
      L     DIW [AR1,P#14.0];
      SLD   3;
      LAR1;
      L     DIB [AR1,P#0.0];
      JU    M083;
M082: +AR1  P#1.0;
      L     DIB [AR1,P#0.0];
      SLW   7;
      LAR2  LD 8;
      +AR2;
      R     DIX [AR2,P#0.0];
      R     DIX [AR2,P#0.1];
      R     DIX [AR2,P#0.2];
      TAK;
M083: LOOP  M082;
      LAR1  LD 0;
      L     DIW [AR1,P#14.0];
      SLD   3;
      LAR2;
      L     B#16#1;
      T     DIB [AR2,P#0.0];
      L     DIB [AR1,P#25.0];
      SLW   3;
      +AR2;
      L     B#16#1;
      T     DIB [AR2,P#0.0];
      TAK;
      +AR2;
      L     B#16#1;
      T     DIB [AR2,P#0.0];
NETWORK
TITLE =
      LAR1  LD 4;
      L     DID [AR1,P#44.0];
      T     LD 8;
      L     DID [AR1,P#80.0];
      LAR2;
      L     DIB [AR2,P#6.0];
      T     LW 22;
      LAR2  LD 0;
      L     DIW [AR2,P#20.0];
      L     DIB [AR2,P#2.0];
      SLW   1;
      +D;
      SLD   3;
      T     LD 24;
      L     DIW [AR2,P#22.0];
      SLD   3;
      T     LD 4;
      L     DIB [LD 8];
      JU    M093;
M084: T     LB 17;
      L     LD 8;
      +     L#8;
      T     LD 8;
      L     DIB [LD 8];
      T     LB 14;
M085: SLW   7;
      LAR1  AR2;
      +AR1;
      +AR1;
      ON    DIX [AR1,P#24.0];
      O     DIX [AR1,P#0.5];
      JC    M092;
      LAR1  LD 4;
      SRW   4;
      +AR1;
      L     LB 14;
      L     DIB [AR1,P#0.0];
      <>I;
      JC    M085;
      LAR1  LD 4;
      SLW   3;
      +AR1;
      L     DIB [AR2,P#3.0];
      SLW   3;
      +AR1;
      +AR1;
      +AR1;
      L     DIB [AR1,P#0.0];
      T     LB 16;
      L     DIW [AR2,P#12.0];
      SLD   3;
      LAR1;
      TAK;
      SLW   7;
      +AR1;
      A     DIX [AR1,P#0.0];
      JC    M092;
      SRW   7;
M086: T     LB 15;
      L     DIW [AR2,P#20.0];
      SLD   3;
      LAR1;
      TAK;
      SLW   3;
      +AR1;
      L     DIB [AR1,P#0.0];
      L     DIB [AR2,P#2.0];
      SLW   5;
      +AR1;
      TAK;
      L     DIB [AR1,P#0.0];
      <>I;
      JC    M087;
      SLW   7;
      LAR1  AR2;
      +AR1;
      +AR1;
      A     DIX [AR1,P#24.0];
      JC    M092;
      JU    M089;
M087: T     LB 14;
M088: SLW   7;
      LAR1  AR2;
      +AR1;
      +AR1;
      A     DIX [AR1,P#24.0];
      JC    M092;
      L     DIB [AR2,P#3.0];
      SLW   3;
      LAR1  LD 4;
      +AR1;
      TAK;
      SRW   4;
      +AR1;
      L     LB 14;
      L     DIB [AR1,P#0.0];
      <>I;
      JC    M088;
M089: LAR1  LD 24;
      L     LB 15;
      SLW   3;
      +AR1;
      L     LB 16;
      L     DIB [AR1,P#0.0];
      <>I;
      JC    M086;
M090: T     LB 15;
      L     DIW [AR2,P#14.0];
      SLD   3;
      LAR1;
      L     LW 22;
      L     DIB [AR1,P#0.0];
      >=I;
      JC    M091;
      L     DID [AR2,P#8.0];
      LAR1;
      S     DIX [AR1,P#26.7];
      JU    M094;
M091: INC   1;
      T     DIB [AR1,P#0.0];
      DEC   1;
      SLW   3;
      +AR1;
      L     LB 15;
      T     DIB [AR1,P#0.0];
      L     DIW [AR2,P#12.0];
      SLD   3;
      LAR1;
      TAK;
      SLW   7;
      +AR1;
      S     DIX [AR1,P#0.0];
      LAR1  LD 24;
      SRW   4;
      +AR1;
      L     LB 16;
      L     DIB [AR1,P#0.0];
      <>I;
      JC    M090;
M092: L     LB 17;
M093: LOOP  M084;
M094: L     DID [AR2,P#8.0];
      T     LD 4;
NETWORK
TITLE =
      LAR1  LD 4;
      CLR;
      A     DIX [AR1,P#13.5];
      =     L 29.7;
      O     DIX [AR1,P#10.6];
      O     DIX [AR1,P#10.7];
      A     L 41.6;
      R     DIX [AR1,P#13.1];
      L     DIW [AR2,P#14.0];
      SLD   3;
      T     LD 8;
      LAR1;
      L     DIB [AR2,P#25.0];
      SLW   3;
      T     LW 22;
      +D;
      T     LD 24;
      L     DIB [AR1,P#0.0];
      T     LB 16;
      SLW   3;
      +AR1;
      L     B#16#0;
      T     DIB [AR1,P#0.0];
      T     LB 15;
      AN    L 29.7;
      JC    M095;
      LAR1  LD 4;
      L     DID [AR1,P#80.0];
      LAR1;
      L     DIB [AR1,P#9.0];
      INC   1;
      T     LB 16;
M095: L     LB 16;
      JU    M101;
M096: T     LB 16;
      LAR1  LD 4;
      L     B#16#0;
      T     DID [AR1,P#72.0];
      L     DID [AR1,P#48.0];
      LAR2;
      A     L 29.7;
      JC    M097;
      L     LD 8;
      +     L#8;
      T     LD 8;
      L     DIB [LD 8];
      JU    M098;
M097: L     LB 15;
      INC   1;
M098: T     LB 15;
      LAR1  LD 0;
      T     DIB [AR1,P#31.0];
      L     B#16#2;
      T     DIB [AR1,P#30.0];
      UC    FB [LW 12];
      LAR1  LD 0;
      L     DIW [AR1,P#12.0];
      SLD   3;
      LAR1;
      L     LB 15;
      SLW   7;
      +AR1;
      =     DIX [AR1,P#0.1];
      LAR2  LD 4;
      AN    DIX [AR1,P#0.0];
      JC    M099;
      O(;
      SRW   7;
      L     DIB [AR2,P#5.0];
      ==I;
      A     L 41.6;
      A     DIX [AR2,P#10.3];
      A     DIX [AR2,P#13.1];
      );
      O(;
      AN    L 41.6;
      A     DIX [AR2,P#10.3];
      A     DIX [AR2,P#13.1];
      );
      R     DIX [AR2,P#13.1];
      S     DIX [AR1,P#0.1];
      L     DID [AR1,P#4.0];
      T     DID [AR1,P#8.0];
M099: L     DID [AR2,P#72.0];
      T     DID [AR1,P#4.0];
      ON    DIX [AR1,P#0.0];
      ON    DIX [AR1,P#0.1];
      JC    M100;
      LAR1  LD 24;
      L     DIB [AR1,P#0.0];
      INC   1;
      T     DIB [AR1,P#0.0];
      DEC   1;
      SLW   3;
      +AR1;
      L     LB 15;
      T     DIB [AR1,P#0.0];
M100: L     LB 16;
M101: LOOP  M096;
NETWORK
TITLE =
// (network holds code this reader does not know; not shown)
NETWORK
TITLE =
// (network holds code this reader does not know; not shown)
NETWORK
TITLE =
      LAR1  LD 0;
      L     DIB [AR1,P#2.0];
      SLW   3;
      L     LD 24;
      +D;
      T     LD 24;
      L     DID [AR1,P#8.0];
      LAR1;
      L     DID [AR1,P#36.0];
      T     LD 4;
      LAR2  LD 8;
      L     DIB [AR2,P#0.0];
      JU    M117;
M113: T     LB 17;
      +AR2  P#1.0;
      LAR1  LD 24;
      L     DIB [AR2,P#0.0];
      T     LB 15;
      SLW   3;
      +AR1;
      L     B#16#0;
      L     DIB [AR1,P#0.0];
      ==I;
      JC    M116;
      T     LB 14;
M114: T     LB 16;
      SLW   7;
      LAR1  LD 0;
      +AR1;
      +AR1;
      O     DIX [AR1,P#0.0];
      O     DIX [AR1,P#1.0];
      JC    M115;
      S     DIX [AR1,P#0.0];
      S     DIX [AR1,P#1.0];
      LAR1  LD 4;
      L     DIB [AR1,P#0.0];
      INC   1;
      T     DIB [AR1,P#0.0];
      DEC   1;
      SLW   3;
      +AR1;
      L     LB 16;
      T     DIB [AR1,P#0.0];
      LAR1  LD 0;
      L     DIW [AR1,P#20.0];
      SLD   3;
      LAR1;
      L     LB 15;
      SLW   3;
      +AR1;
      L     DIB [AR1,P#0.0];
      L     B#16#0;
      <>I;
      JC    M116;
M115: LAR1  LD 0;
      L     DIW [AR1,P#22.0];
      L     DIB [AR1,P#3.0];
      +D;
      SLD   3;
      LAR1;
      L     LB 16;
      SLW   3;
      +AR1;
      L     LB 14;
      L     DIB [AR1,P#0.0];
      <>I;
      JC    M114;
M116: L     LB 17;
M117: LOOP  M113;
NETWORK
TITLE =
      LAR1  LD 4;
      LAR2  LD 0;
      L     DID [AR2,P#8.0];
      T     LD 4;
      L     B#16#2;
      JU    M251;
M118: NOP   0;
NETWORK
TITLE =
      LAR1  LD 8;
      LAR2  LD 4;
      L     B#16#1;
      L     DIB [AR1,P#0.0];
      <I;
      A     DIX [AR2,P#11.3];
      JC    M081;
NETWORK
TITLE =
      L     DID [AR2,P#44.0];
      LAR1;
      L     DIB [AR1,P#0.0];
      JU    M120;
M119: +AR1  P#1.0;
      L     DIB [AR1,P#0.0];
      SLW   7;
      LAR2  LD 0;
      +AR2;
      +AR2;
      R     DIX [AR2,P#24.0];
      TAK;
M120: LOOP  M119;
NETWORK
TITLE =
      LAR1  LD 4;
      L     DID [AR1,P#80.0];
      LAR2;
      AN    DIX [AR2,P#34.7];
      JC    M129;
      L     DIW [AR2,P#32.0];
      T     LW 18;
      L     B#16#2;
      -D;
      SLD   3;
      LAR2;
      L     DIW [AR2,P#0.0];
      T     LW 20;
      L     LW 18;
      LAR2  LD 0;
      L     DIB [AR2,P#3.0];
      INC   2;
      -D;
      SLD   3;
      T     LD 8;
      L     DIB [LD 8];
      T     LW 18;
      L     DID [AR1,P#36.0];
      T     LD 24;
      L     DIB [LD 24];
      JU    M128;
M121: T     LB 17;
      L     LD 24;
      +     L#8;
      T     LD 24;
      L     DIB [LD 24];
      SLW   3;
      LAR1  LD 8;
      +AR1;
      L     DIB [AR1,P#0.0];
      T     LW 22;
      SET;
      =     L 29.6;
      LAR1  LD 0;
      L     DID [AR1,P#4.0];
      LAR2;
M122: L     DIB [AR2,P#0.0];
      JU    M126;
M123: T     LB 14;
      +AR2  P#1.0;
      L     DIB [LD 24];
      L     DIB [AR2,P#0.0];
      <>I;
      JC    M124;
      A     L 29.6;
      JC    M125;
      L     B#16#1;
      T     LB 14;
      JC    M125;
M124: T     LB 16;
      SLW   3;
      LAR1  LD 8;
      +AR1;
      L     DIB [AR1,P#0.0];
      L     LW 18;
      *D;
      L     LW 22;
      +D;
      L     LW 20;
      SLD   3;
      +D;
      LAR1;
      A     DIX [AR1,P#0.0];
      JC    M125;
      L     LB 16;
      SLW   7;
      LAR1  LD 0;
      +AR1;
      +AR1;
      O     DIX [AR1,P#0.5];
      ON    DIX [AR1,P#1.0];
      JC    M125;
      S     DIX [AR1,P#0.5];
      R     DIX [AR1,P#1.0];
      LAR1  LD 4;
      L     DID [AR1,P#40.0];
      LAR1;
      L     DIB [AR1,P#0.0];
      INC   1;
      T     DIB [AR1,P#0.0];
      DEC   1;
      SLW   3;
      +AR1;
      L     LB 16;
      T     DIB [AR1,P#0.0];
M125: L     LB 14;
M126: LOOP  M123;
      AN    L 29.6;
      JC    M127;
      R     L 29.6;
      LAR1  LD 4;
      L     DID [AR1,P#36.0];
      LAR2;
      JU    M122;
M127: L     LB 17;
M128: LOOP  M121;
M129: NOP   0;
NETWORK
TITLE =
      LAR1  LD 4;
      L     DID [AR1,P#40.0];
      LAR1;
      L     B#16#2;
      JU    M270;
M130: NOP   0;
NETWORK
TITLE =
      LAR1  LD 4;
      L     DID [AR1,P#36.0];
      T     LD 8;
      LAR1;
      L     B#16#1;
      JU    M270;
M131: NOP   0;
NETWORK
TITLE =
      LAR1  LD 8;
      L     DIB [AR1,P#0.0];
      JU    M133;
M132: T     LB 14;
      +AR1  P#1.0;
      L     DIB [AR1,P#0.0];
      SLW   7;
      LAR2  LD 0;
      +AR2;
      +AR2;
      L     B#16#0;
      T     DID [AR2,P#4.0];
      T     DID [AR2,P#8.0];
      L     LB 14;
M133: LOOP  M132;
NETWORK
TITLE =
      LAR1  LD 0;
      L     DID [AR1,P#4.0];
      T     LD 8;
      LAR2;
      LAR1  LD 4;
      L     DID [AR1,P#44.0];
      LAR1;
      L     DIB [AR2,P#0.0];
M134: L     DIB [AR2,P#0.0];
      T     DIB [AR1,P#0.0];
      +AR1  P#1.0;
      +AR2  P#1.0;
      TAK;
      LOOP  M134;
      LAR1  LD 4;
      SET;
      S     DIX [AR1,P#27.6];
      LAR1  LD 8;
      L     B#16#0;
      JU    M270;
M135: NOP   0;
NETWORK
TITLE =
      LAR1  LD 4;
      L     DID [AR1,P#80.0];
      LAR2;
      L     DIB [AR2,P#7.0];
      T     LB 14;
      L     DID [AR1,P#36.0];
      LAR1;
      L     DIB [AR1,P#0.0];
      DEC   1;
      LAR2  LD 8;
      L     DIB [AR2,P#0.0];
      DEC   1;
      +I;
      L     LB 14;
      <=I;
      JC    M137;
      LAR2  LD 4;
      S     DIX [AR2,P#26.6];
      -I;
      T     LB 14;
      L     DIB [AR1,P#0.0];
      TAK;
      -I;
      T     DIB [AR1,P#0.0];
      SLW   3;
      +AR1;
      L     LB 14;
M136: T     LB 14;
      L     DIB [AR1,P#0.0];
      SLW   7;
      LAR2  LD 0;
      +AR2;
      +AR2;
      L     B#16#0;
      T     DIW [AR2,P#0.0];
      +AR1  P#1.0;
      L     LB 14;
      LOOP  M136;
M137: NOP   0;
NETWORK
TITLE =
// (network holds code this reader does not know; not shown)
NETWORK
TITLE =
      LAR1  LD 0;
      L     DIW [AR1,P#16.0];
      L     DIB [AR1,P#26.0];
      +D;
      SLD   3;
      LAR1;
      LAR2  LD 4;
      L     DID [AR2,P#40.0];
      LAR2;
      L     DIB [AR2,P#0.0];
M170: L     DIB [AR2,P#0.0];
      T     DIB [AR1,P#0.0];
      +AR1  P#1.0;
      +AR2  P#1.0;
      TAK;
      LOOP  M170;
      LAR1  LD 4;
      L     DID [AR1,P#36.0];
      LAR1;
      LAR2  LD 0;
      L     DID [AR2,P#4.0];
      LAR2;
      L     DIB [AR2,P#0.0];
      T     LB 14;
      L     DIB [AR1,P#0.0];
      DEC   1;
      +I;
      T     DIB [AR2,P#0.0];
      L     LB 14;
      SLW   3;
      +AR2;
      L     DIB [AR1,P#0.0];
      JU    M172;
M171: +AR1  P#1.0;
      L     DIB [AR1,P#0.0];
      T     DIB [AR2,P#0.0];
      +AR2  P#1.0;
      TAK;
M172: LOOP  M171;
      LAR1  LD 4;
      SET;
      R     DIX [AR1,P#27.6];
NETWORK
TITLE =
      LAR1  LD 0;
      L     B#16#6;
      T     DIB [AR1,P#30.0];
      LAR1  LD 4;
      L     DID [AR1,P#48.0];
      LAR2;
      UC    FB [LW 12];
      LAR1  LD 4;
      SET;
      R     DIX [AR1,P#27.5];
NETWORK
TITLE =
      LAR1  LD 0;
      L     DIW [AR1,P#18.0];
      SLD   3;
      T     LD 8;
      LAR1  LD 4;
      SET;
      R     DIX [AR1,P#26.1];
      R     DIX [AR1,P#26.2];
      L     DIB [LD 8];
      JU    M174;
M173: T     LB 14;
      L     LD 8;
      +     L#8;
      T     LD 8;
      L     DIB [LD 8];
      SLW   7;
      LAR2  LD 0;
      +AR2;
      +AR2;
      A     DIX [AR2,P#1.1];
      S     DIX [AR1,P#26.1];
      A     DIX [AR2,P#1.2];
      S     DIX [AR1,P#26.2];
      L     LB 14;
M174: LOOP  M173;
      O     DIX [AR1,P#26.1];
      O     DIX [AR1,P#26.2];
      =     DIX [AR1,P#26.0];
      O     DIX [AR1,P#26.4];
      O     DIX [AR1,P#26.5];
      O     DIX [AR1,P#26.6];
      O     DIX [AR1,P#26.7];
      O     DIX [AR1,P#27.0];
      =     DIX [AR1,P#26.3];
NETWORK
TITLE =
// (network holds code this reader does not know; not shown)
NETWORK
TITLE =
      CLR;
      AN    DIX [AR1,P#26.3];
      SAVE;
      L     DID [AR1,P#48.0];
      LAR2;
      BE;
NETWORK
TITLE =
M251: T     LB 28;
      LAR2  LD 4;
      L     DID [AR2,P#44.0];
      T     LD 24;
      CLR;
      L     DIB [AR1,P#0.0];
      JU    M254;
M252: T     LB 17;
      +AR1  P#1.0;
      L     DIB [AR1,P#0.0];
      SLW   7;
      LAR2  LD 0;
      +AR2;
      +AR2;
      A     DIX [AR2,P#24.0];
      JC    M253;
      S     DIX [AR2,P#24.0];
      LAR2  LD 24;
      L     DIB [AR2,P#0.0];
      INC   1;
      T     DIB [AR2,P#0.0];
      DEC   1;
      SLW   3;
      +AR2;
      TAK;
      SRW   7;
      T     DIB [AR2,P#0.0];
M253: L     LB 17;
M254: LOOP  M252;
      L     LB 28;
      JL    M255;
      JU    M048;
      JU    M055;
      JU    M118;
M255: NOP   0;
NETWORK
TITLE =
M256: T     LB 28;
      LAR2  LD 4;
      L     DID [AR2,P#36.0];
      T     LD 24;
      CLR;
      L     DIB [AR1,P#0.0];
      JU    M259;
M257: T     LB 17;
      +AR1  P#1.0;
      L     DIB [AR1,P#0.0];
      SLW   7;
      LAR2  LD 0;
      +AR2;
      +AR2;
      O     DIX [AR2,P#0.0];
      O     DIX [AR2,P#1.0];
      JC    M258;
      S     DIX [AR2,P#0.0];
      S     DIX [AR2,P#1.0];
      LAR2  LD 24;
      L     DIB [AR2,P#0.0];
      INC   1;
      T     DIB [AR2,P#0.0];
      DEC   1;
      SLW   3;
      +AR2;
      TAK;
      SRW   7;
      T     DIB [AR2,P#0.0];
M258: L     LB 17;
M259: LOOP  M257;
      L     LB 28;
      JL    M260;
      JU    M052;
      JU    M071;
M260: NOP   0;
NETWORK
TITLE =
M261: T     LB 28;
      LAR2  LD 4;
      L     DID [AR2,P#40.0];
      T     LD 24;
      CLR;
      L     DIB [AR1,P#0.0];
      JU    M264;
M262: T     LB 17;
      +AR1  P#1.0;
      L     DIB [AR1,P#0.0];
      SLW   7;
      LAR2  LD 0;
      +AR2;
      +AR2;
      O     DIX [AR2,P#0.5];
      ON    DIX [AR2,P#1.0];
      JC    M263;
      S     DIX [AR2,P#0.5];
      R     DIX [AR2,P#1.0];
      LAR2  LD 24;
      L     DIB [AR2,P#0.0];
      INC   1;
      T     DIB [AR2,P#0.0];
      DEC   1;
      SLW   3;
      +AR2;
      TAK;
      SRW   7;
      T     DIB [AR2,P#0.0];
M263: L     LB 17;
M264: LOOP  M262;
      L     LB 28;
      JL    M265;
      JU    M049;
      JU    M051;
      JU    M074;
M265: NOP   0;
NETWORK
TITLE =
M266: T     LB 28;
      TAK;
      T     LW 20;
      L     B#16#0;
      T     LW 18;
      L     DID [AR1,P#80.0];
      LAR2;
      L     DIB [AR2,P#12.0];
      LAR2  LD 0;
M267: T     LB 17;
      L     LW 18;
      INC   1;
      T     LW 18;
      +AR2  P#32.0;
      L     LW 20;
      L     DIW [AR2,P#2.0];
      ==I;
      L     LW 18;
      JC    M268;
      L     LB 17;
      LOOP  M267;
      S     DIX [AR1,P#26.4];
M268: L     LB 28;
      JL    M269;
      JU    M069;
      JU    M072;
      JU    M067;
M269: NOP   0;
NETWORK
TITLE =
M270: T     LB 28;
      CLR;
      TAR1  LD 24;
      L     DIB [AR1,P#0.0];
      L     B#16#1;
      T     DIB [AR1,P#0.0];
      TAK;
      JU    M278;
M271: T     LB 17;
      +AR1  P#1.0;
      L     DIB [AR1,P#0.0];
      SLW   7;
      LAR2  LD 0;
      +AR2;
      +AR2;
      L     LB 28;
      JL    M272;
      JU    M273;
      JU    M275;
      JU    M274;
      JU    M275;
      JU    M274;
M272: NOP   0;
M273: A     DIX [AR2,P#0.5];
      JC    M277;
      JU    M276;
M274: A     DIX [AR2,P#0.5];
      A     DIX [AR2,P#0.0];
      R     DIX [AR2,P#0.5];
      R     DIX [AR2,P#0.0];
      JC    M277;
      JU    M276;
M275: AN    DIX [AR2,P#0.0];
      JC    M277;
M276: LAR2  LD 24;
      L     DIB [AR2,P#0.0];
      INC   1;
      T     DIB [AR2,P#0.0];
      DEC   1;
      SLW   3;
      +AR2;
      L     DIB [AR1,P#0.0];
      T     DIB [AR2,P#0.0];
M277: L     LB 17;
M278: LOOP  M271;
      L     LB 28;
      JL    M279;
      JU    M135;
      JU    M131;
      JU    M130;
      JU    M054;
      JU    M053;
M279: NOP   0;
NETWORK
TITLE =
M280: CLR;
      LAR1  LD 0;
      L     DIW [AR1,P#18.0];
      SLD   3;
      T     LD 24;
      LAR2;
      LAR1;
      L     DIB [AR1,P#0.0];
      JU    M284;
M281: T     LB 17;
      +AR1  P#1.0;
      L     LB 14;
      L     DIB [AR1,P#0.0];
      <>I;
      JC    M282;
      L     DIB [LD 24];
      DEC   1;
      T     DIB [LD 24];
      JU    M283;
M282: +AR2  P#1.0;
      T     DIB [AR2,P#0.0];
M283: L     LB 17;
M284: LOOP  M281;
      A     L 29.0;
      JC    M162;
      JU    M150;
NETWORK
TITLE =
M285: L     DIB [AR1,P#0.0];
      JU    M287;
M286: T     LB 17;
      +AR1  P#1.0;
      L     DIB [AR1,P#0.0];
      SLW   7;
      LAR2  LD 0;
      +AR2;
      +AR2;
      L     B#16#0;
      T     DIB [AR2,P#0.0];
      L     LB 17;
M287: LOOP  M286;
      CLR;
      A     L 29.0;
      JC    M047;
      JU    M046;
NETWORK
TITLE =
M288: T     LW 20;
      LAR1  LD 4;
      L     DID [AR1,P#68.0];
      LAR1;
      CLR;
      A     L 29.0;
      JC    M289;
      LAR2  LD 0;
      L     DIB [AR2,P#26.0];
      SLW   3;
      +AR1;
M289: LAR2  LD 4;
      L     DID [AR2,P#80.0];
      LAR2;
      L     DIB [AR2,P#7.0];
      L     DIB [AR1,P#0.0];
      <I;
      LAR2  LD 4;
      S     DIX [AR2,P#26.5];
      JC    M290;
      INC   1;
      T     DIB [AR1,P#0.0];
      DEC   1;
      SLW   3;
      +AR1;
      L     LW 20;
      T     DIB [AR1,P#0.0];
M290: A     L 29.0;
      JC    M073;
      JU    M070;
NETWORK
TITLE =
// (network holds code this reader does not know; not shown)
NETWORK
TITLE =
M318: L     DINO;
      L     DID [AR1,P#52.0];
      +D;
      T     DID [AR1,P#52.0];
      SRD   16;
      T     LW 12;
      BLD   7;
      UC    "TIME_TCK";
      {     P#L 8.0 };
      BLD   8;
      L     LD 8;
      T     DID [AR1,P#18.0];
      L     LD 24;
      T     DID [AR1,P#80.0];
      LAR2;
      L     DID [AR1,P#48.0];
      AD    DW#16#7FFFF;
      T     LD 8;
      L     DID [AR1,P#36.0];
      +D;
      T     DID [AR1,P#36.0];
      TAK;
      L     DID [AR1,P#40.0];
      +D;
      T     DID [AR1,P#40.0];
      TAK;
      L     DID [AR1,P#44.0];
      +D;
      T     DID [AR1,P#44.0];
      TAK;
      L     DID [AR1,P#68.0];
      +D;
      T     DID [AR1,P#68.0];
      TAK;
      L     DID [AR1,P#28.0];
      +D;
      T     DID [AR1,P#28.0];
      T     LD 0;
      LAR1;
      A     L 29.1;
      JC    M321;
      L     W#16#FB;
      L     DIW [AR2,P#30.0];
      ==I;
      JC    M320;
      L     W#16#FC;
      ==I;
      JC    M319;
      L     DW#16#40000000;
      T     DID [AR2,P#14.0];
      L     DW#16#0;
      T     DID [AR2,P#18.0];
      L     B#16#2;
      JU    M322;
M319: L     DW#16#E000F6C8;
      T     DID [AR2,P#14.0];
      L     DW#16#E000800D;
      T     DID [AR2,P#18.0];
      L     B#16#A;
      JU    M322;
M320: L     DW#16#E3E0F6C8;
      T     DID [AR2,P#14.0];
      L     DW#16#E000BE0D;
      T     DID [AR2,P#18.0];
      L     B#16#A;
      JU    M322;
M321: L     DIW [AR2,P#32.0];
M322: L     LD 8;
      SRD   3;
      +D;
      T     DIW [AR1,P#12.0];
      TAR1;
      SRD   3;
      L     DIB [AR2,P#12.0];
      T     LB 14;
      INC   1;
      SLW   5;
      +D;
      L     DIW [AR2,P#0.0];
      SLD   2;
      +D;
      L     DIW [AR2,P#2.0];
      SLD   2;
      +D;
      T     DIW [AR1,P#14.0];
      L     DIB [AR2,P#9.0];
      T     LB 15;
      INC   2;
      SRW   1;
      SLW   1;
      T     DIB [AR1,P#2.0];
      L     LB 14;
      INC   2;
      SRW   1;
      SLW   1;
      T     DIB [AR1,P#3.0];
      L     DIB [AR2,P#6.0];
      INC   3;
      SRW   1;
      SLW   1;
      T     DIB [AR1,P#25.0];
      L     DIB [AR2,P#7.0];
      INC   3;
      SRW   1;
      SLW   1;
      T     DIB [AR1,P#26.0];
      L     LB 14;
      INC   3;
      SRW   1;
      SLW   1;
      T     DIB [AR1,P#27.0];
      L     LD 4;
      T     DID [AR1,P#8.0];
      L     DIW [AR1,P#14.0];
      L     DIB [AR1,P#25.0];
      SLW   1;
      +D;
      T     DIW [AR1,P#16.0];
      L     DIB [AR1,P#26.0];
      SLW   2;
      +D;
      SLD   3;
      T     DID [AR1,P#4.0];
      SRD   3;
      L     DIB [AR1,P#26.0];
      +D;
      T     DIW [AR1,P#18.0];
      TAR2;
      SRD   3;
      L     DIB [AR1,P#3.0];
      SLW   2;
      -D;
      T     DIW [AR1,P#22.0];
      L     DIB [AR1,P#2.0];
      SLW   2;
      -D;
      L     DIB [AR1,P#2.0];
      -D;
      T     DIW [AR1,P#20.0];
      L     DIB [AR1,P#26.0];
      -D;
      T     DIW [AR1,P#28.0];
      A     L 29.1;
      JC    M323;
      L     DIW [AR2,P#32.0];
      JU    M324;
M323: L     DIW [AR2,P#28.0];
M324: L     W#16#105;
      ==I;
      JC    M325;
      TAK;
      L     W#16#107;
      <>I;
      JC    M328;
M325: L     DIW [AR1,P#12.0];
      SLD   3;
      LAR2;
      L     B#16#0;
      L     LB 14;
M326: +AR1  P#32.0;
      TAK;
      INC   1;
      T     DIB [AR1,P#3.0];
      S     DIX [AR1,P#1.6];
      TAK;
      LOOP  M326;
      L     LB 15;
M327: +AR2  P#16.0;
      TAK;
      INC   1;
      T     DIB [AR2,P#3.0];
      S     DIX [AR2,P#0.3];
      TAK;
      LOOP  M327;
      LAR1  LD 0;
      L     B#16#7;
      T     DIB [AR1,P#30.0];
      LAR1  LD 4;
      L     DID [AR1,P#48.0];
      LAR2;
      UC    FB [LW 12];
M328: LAR1  LD 4;
      SET;
      S     DIX [AR1,P#27.2];
      JU    M005;
NETWORK
TITLE =
// (network holds code this reader does not know; not shown)
END_FUNCTION

